IF L_Runtime_OK AND (GVL_TIME_MONOTONIC.Boot_Generation_ID = 0) THEN
    L_Runtime_OK := FALSE;
    L_Error_Code := 4905;
    L_Error_Text := 'Boot generation missing';
END_IF;

IF L_Runtime_OK AND (NOT GVL_STATUS.G_Is_Active_PLC) THEN
    L_Runtime_OK := FALSE;
    L_Error_Code := 5000;
    L_Error_Text := 'Runtime barrier inactive PLC';
END_IF;

IF L_Runtime_OK AND (NOT GVL_PLC_FENCING.PLC_Ownership_Valid) THEN
    L_Runtime_OK := FALSE;
    L_Error_Code := 5010;
    L_Error_Text := 'PLC ownership invalid';
END_IF;

IF L_Runtime_OK AND (NOT GVL_PLC_FENCING.PLC_Semantic_Authority_Valid) THEN
    L_Runtime_OK := FALSE;
    L_Error_Code := 5011;
    L_Error_Text := 'PLC semantic authority invalid';
END_IF;

IF L_Runtime_OK AND GVL_PLC_FENCING.PLC_Forced_Safe_Quarantine THEN
    L_Runtime_OK := FALSE;
    L_Error_Code := 5012;
    L_Error_Text := 'PLC fencing quarantine active';
END_IF;

IF L_Runtime_OK AND GVL_PLC_FENCING.PLC_Lease_Expired THEN
    L_Runtime_OK := FALSE;
    L_Error_Code := 5013;
    L_Error_Text := 'PLC authority lease expired';
END_IF;

IF L_Runtime_OK AND (GVL_PLC_FENCING.PLC_Fencing_Token = 0) THEN
    L_Runtime_OK := FALSE;
    L_Error_Code := 5014;
    L_Error_Text := 'PLC fencing token missing';
END_IF;

IF L_Runtime_OK AND (NOT GVL_TRANSPORT_FRESHNESS.Transport_Freshness_Valid) THEN
    L_Runtime_OK := FALSE;
    L_Error_Code := 5200;
    L_Error_Text := 'Transport freshness invalid';
END_IF;

IF L_Runtime_OK AND (NOT GVL_TRANSPORT_FRESHNESS.Transport_Publication_Allowed) THEN
    L_Runtime_OK := FALSE;
    L_Error_Code := 5201;
    L_Error_Text := 'Transport publication blocked';
END_IF;

IF L_Runtime_OK AND GVL_TRANSPORT_FRESHNESS.Transport_Quarantine_Active THEN
    L_Runtime_OK := FALSE;
    L_Error_Code := 5202;
    L_Error_Text := 'Transport quarantine active';
END_IF;

IF L_Runtime_OK AND GVL_TRANSPORT_FRESHNESS.Transport_Lease_Expired THEN
    L_Runtime_OK := FALSE;
    L_Error_Code := 5203;
    L_Error_Text := 'Transport lease expired';
END_IF;

IF L_Runtime_OK AND GVL_TRANSPORT_FRESHNESS.Transport_Snapshot_Invalid THEN
    L_Runtime_OK := FALSE;
    L_Error_Code := 5204;
    L_Error_Text := 'Transport snapshot invalid';
END_IF;

// Finalized distributed commit continuity.
// Intentionally excludes semantic continuity
// to avoid primordial semantic/runtime recursion.
L_Finalized_Continuity_Healthy :=
    GVL_DISTRIBUTED_SNAPSHOT.Distributed_Publication_Reconciled
    AND GVL_DISTRIBUTED_SNAPSHOT.Distributed_Publication_Freeze_Valid
    AND GVL_DISTRIBUTED_SNAPSHOT.Distributed_Snapshot_Consistent
    AND GVL_DISTRIBUTED_COMMIT.Distributed_Commit_Valid
    AND GVL_DISTRIBUTED_COMMIT.Publication_Prepare_Valid
    AND GVL_DISTRIBUTED_COMMIT.Publication_Commit_Confirmed
    AND NOT GVL_DISTRIBUTED_COMMIT.Peer_Commit_Mismatch
    AND NOT GVL_DISTRIBUTED_COMMIT.Commit_Lease_Expired;

IF L_Runtime_OK
AND NOT L_Finalized_Continuity_Healthy THEN
    L_Runtime_OK := FALSE;
    L_Error_Code := 5300;
    L_Error_Text := 'Finalized continuity invalid';
END_IF;

IF L_Runtime_OK THEN
    IF (GVL_SAFETY_SHUTDOWN.G_Safety_Mode = FIRE)
    AND (GVL_COMMAND_SHADOW.G_Vent_Stop)
    THEN
        L_Runtime_OK := FALSE;
        L_Error_Code := 5003;
        L_Error_Text := 'Impossible fire ventilation state';
    END_IF;
END_IF;

IF L_Runtime_OK THEN
    IF (GVL_SAFETY_SHUTDOWN.G_Safety_Mode = GAS)
    AND (NOT GVL_COMMAND_SHADOW.G_Gas_Valve_Close)
    THEN
        L_Runtime_OK := FALSE;
        L_Error_Code := 5004;
        L_Error_Text := 'Impossible gas valve state';
    END_IF;
END_IF;

GVL_RUNTIME_EPOCH.Runtime_Runtime_Barrier_OK := L_Runtime_OK;
GVL_RUNTIME_EPOCH.Runtime_Snapshot_Valid := L_Runtime_OK;
GVL_RUNTIME_EPOCH.Runtime_PLC_Authority_Valid :=
    GVL_STATUS.G_Is_Active_PLC
    AND GVL_PLC_FENCING.PLC_Semantic_Authority_Valid
    AND GVL_PLC_FENCING.PLC_Ownership_Valid
    AND GVL_TIME_MONOTONIC.Monotonic_Time_Valid
    AND GVL_TRANSPORT_FRESHNESS.Transport_Freshness_Valid
    AND L_Finalized_Continuity_Healthy;

GVL_RUNTIME_EPOCH.Runtime_Last_Validation_Time_MS := L_Now_MS;

IF L_Runtime_OK THEN
    GVL_RUNTIME_EPOCH.Runtime_Epoch := GVL_RUNTIME_EPOCH.Runtime_Epoch + 1;
    GVL_RUNTIME_EPOCH.Runtime_IO_Publication_Allowed := TRUE;
    GVL_RUNTIME_EPOCH.Runtime_Snapshot_Published := TRUE;
    GVL_RUNTIME_EPOCH.Runtime_Last_Error_Code := 0;
    GVL_RUNTIME_EPOCH.Runtime_Last_Error_Text := '';
ELSE
    GVL_RUNTIME_EPOCH.Runtime_Impossible_State_Detected := TRUE;
    GVL_RUNTIME_EPOCH.Runtime_Last_Error_Code := L_Error_Code;
    GVL_RUNTIME_EPOCH.Runtime_Last_Error_Text := L_Error_Text;
    GVL_RUNTIME_EPOCH.Runtime_Barrier_Block_Count := GVL_RUNTIME_EPOCH.Runtime_Barrier_Block_Count + 1;
END_IF;

GVL_RUNTIME_EPOCH.Runtime_Cycle_End_MS := L_Now_MS;
          
END_PROGRAM

PROGRAM PRG_Distributed_Epoch_Linearity_Governor

            IF GVL_TEMPORAL_CAUSALITY_CLOSURE_FABRIC.Temporal_Causality_Closure_Granted
AND NOT GVL_DISTRIBUTED_EPOCH_LINEARITY_FABRIC.Epoch_Rollback_Detected
AND NOT GVL_DISTRIBUTED_EPOCH_LINEARITY_FABRIC.Distributed_Epoch_Fork_Detected
AND NOT GVL_DISTRIBUTED_EPOCH_LINEARITY_FABRIC.Stale_Epoch_Application_Detected THEN

    GVL_DISTRIBUTED_EPOCH_LINEARITY_FABRIC.Distributed_Epoch_Linearity_Valid := TRUE;
    GVL_DISTRIBUTED_EPOCH_LINEARITY_FABRIC.Distributed_Epoch_Linearity_Granted := TRUE;
    GVL_DISTRIBUTED_EPOCH_LINEARITY_FABRIC.Distributed_Epoch_Linearity_Valid_Proof := TRUE;
    GVL_DISTRIBUTED_EPOCH_LINEARITY_FABRIC.Epoch_Timeline_Monotonic := TRUE;
    GVL_DISTRIBUTED_EPOCH_LINEARITY_FABRIC.Cluster_Epoch_Consensus_Stable := TRUE;
END_IF;
          
END_PROGRAM

PROGRAM PRG_PLC_Fencing_Governor
  VAR
    L_Now_MS : UDINT;
    L_Delta_MS : UDINT;
    L_Authority_Valid : BOOL := TRUE;
    L_Error_Code : UDINT := 0;
    L_Error_Text : STRING(160) := '';
  END_VAR

            L_Now_MS := GVL_STATUS.G_System_Time_MS;
L_Authority_Valid := TRUE;
L_Error_Code := 0;
L_Error_Text := '';

// ======================================================
// PLC FENCING GOVERNOR
// ======================================================
// Governs distributed PLC ownership semantics.
// Prevents stale-owner resurrection and split-brain.
// ======================================================

GVL_PLC_FENCING.PLC_Split_Brain_Detected := FALSE;
GVL_PLC_FENCING.PLC_Stale_Owner_Detected := FALSE;
GVL_PLC_FENCING.PLC_Asymmetric_Partition_Detected := FALSE;
GVL_PLC_FENCING.PLC_Forced_Safe_Quarantine := FALSE;

// Active PLC ownership validation.
IF L_Authority_Valid AND (NOT GVL_STATUS.G_Is_Active_PLC) THEN
    L_Authority_Valid := FALSE;
    L_Error_Code := 7001;
    L_Error_Text := 'PLC ownership inactive';
END_IF;

// Lease freshness validation.
L_Delta_MS := L_Now_MS - GVL_PLC_FENCING.PLC_Last_Lease_Refresh_MS;

IF L_Authority_Valid AND GVL_PLC_FENCING.PLC_Lease_Active THEN
    IF L_Delta_MS > GVL_PLC_FENCING.PLC_Lease_Timeout_MS THEN
        L_Authority_Valid := FALSE;
        L_Error_Code := 7002;
        L_Error_Text := 'PLC lease expired';
    END_IF;
END_IF;

// Heartbeat-only ownership is unsafe.
IF L_Authority_Valid AND GVL_PLC_FENCING.PLC_Heartbeat_Only_Mode THEN
    L_Authority_Valid := FALSE;
    L_Error_Code := 7003;
    L_Error_Text := 'Heartbeat-only ownership rejected';
END_IF;

// Publish authoritative fencing state.
IF L_Authority_Valid THEN
    GVL_PLC_FENCING.PLC_Ownership_Epoch := GVL_PLC_FENCING.PLC_Ownership_Epoch + 1;
    GVL_PLC_FENCING.PLC_Fencing_Token := GVL_PLC_FENCING.PLC_Ownership_Epoch;

    GVL_PLC_FENCING.PLC_Ownership_Valid := TRUE;
    GVL_PLC_FENCING.PLC_Semantic_Authority_Valid := TRUE;

    GVL_PLC_FENCING.PLC_Lease_Active := TRUE;
    GVL_PLC_FENCING.PLC_Lease_Expired := FALSE;

    GVL_PLC_FENCING.PLC_Last_Lease_Refresh_MS := L_Now_MS;
    GVL_PLC_FENCING.PLC_Last_Authority_Validation_MS := L_Now_MS;

    GVL_PLC_FENCING.PLC_Last_Error_Code := 0;
    GVL_PLC_FENCING.PLC_Last_Error_Text := '';
ELSE
    GVL_PLC_FENCING.PLC_Ownership_Valid := FALSE;
    GVL_PLC_FENCING.PLC_Semantic_Authority_Valid := FALSE;

    GVL_PLC_FENCING.PLC_Lease_Expired := TRUE;
    GVL_PLC_FENCING.PLC_Forced_Safe_Quarantine := TRUE;

    GVL_PLC_FENCING.PLC_Last_Error_Code := L_Error_Code;
    GVL_PLC_FENCING.PLC_Last_Error_Text := L_Error_Text;

    IF L_Error_Code = 7002 THEN
        GVL_PLC_FENCING.PLC_Stale_Owner_Detected := TRUE;
    END_IF;

    IF L_Error_Code = 7003 THEN
        GVL_PLC_FENCING.PLC_Split_Brain_Detected := TRUE;
        GVL_PLC_FENCING.PLC_Asymmetric_Partition_Detected := TRUE;
    END_IF;

    GVL_PLC_FENCING.PLC_Fencing_Invalidation_Count := GVL_PLC_FENCING.PLC_Fencing_Invalidation_Count + 1;
END_IF;
          
END_PROGRAM

PROGRAM PRG_IO_Read
  VAR
    L_i : INT;
    L_Map_Index : INT;
    L_Glass_Index : INT;
    L_Debounce_Time : TIME := T#100MS;
    L_Manifold_Pressure_Raw : WORD;
    L_Manifold_Current_Raw : WORD;
    L_Filtered_Room_Temp : REAL;
    L_Filtered_Floor_Temp : REAL;
    fbDebounce_Switches : ARRAY[1..GVL_CONSTANTS.C_MAX_LIGHT_ZONES] OF FB_System_Timer;
    fbDebounce_Motion : ARRAY[1..GVL_CONSTANTS.C_MAX_LIGHT_ZONES] OF FB_System_Timer;
    fbDebounce_Security_Open : ARRAY[1..GVL_CONSTANTS.C_MAX_SECURITY_SENSORS] OF FB_System_Timer;
    fbDebounce_Security_Glass : ARRAY[1..GVL_CONSTANTS.C_MAX_SECURITY_SENSORS] OF FB_System_Timer;
    fbDebounce_Flood : ARRAY[1..GVL_CONSTANTS.C_MAX_FLOOD_SENSORS] OF FB_System_Timer;
    fbDebounce_Smoke : ARRAY[1..GVL_CONSTANTS.C_MAX_SMOKE_SENSORS] OF FB_System_Timer;
    fbDebounce_Group_2F : FB_System_Timer;
    fbIO_Watchdog_1 : FB_IO_Module_Watchdog;
    fbIO_Watchdog_2 : FB_IO_Module_Watchdog;
    fbDiagEventManager : FB_Diagnostics_Event_Manager;
    L_IO_Error_Active : BOOL;
    fbCalib_Outdoor_Temp : FB_Sensor_Calibration_Processor;
    fbCalib_Supply_Temps : ARRAY[1..GVL_CONSTANTS.C_MAX_SUPPLY_TEMPS] OF FB_Sensor_Calibration_Processor;
    fbCalib_Room_Temps : ARRAY[1..GVL_CONSTANTS.C_MAX_ZONES] OF FB_Sensor_Calibration_Processor;
    fbCalib_Floor_Temps : ARRAY[1..GVL_CONSTANTS.C_MAX_ZONES] OF FB_Sensor_Calibration_Processor;
    fbCalib_Room_Hum : ARRAY[1..GVL_CONSTANTS.C_MAX_ZONES] OF FB_Sensor_Calibration_Processor;
    fbCalib_Room_CO2 : ARRAY[1..GVL_CONSTANTS.C_MAX_ZONES] OF FB_Sensor_Calibration_Processor;
    fbCalib_Manifold_T_Supply : ARRAY[1..GVL_CONSTANTS.C_MAX_MANIFOLDS] OF FB_Sensor_Calibration_Processor;
    fbCalib_Manifold_T_Return : ARRAY[1..GVL_CONSTANTS.C_MAX_MANIFOLDS] OF FB_Sensor_Calibration_Processor;
    fbCalib_Methane : ARRAY[1..GVL_CONSTANTS.C_MAX_METHANE_SENSORS] OF FB_Sensor_Calibration_Processor;
    fbCalib_CO : ARRAY[1..GVL_CONSTANTS.C_MAX_CO_SENSORS] OF FB_Sensor_Calibration_Processor;
    fbAnalog_Manifold_Pressure : ARRAY[1..GVL_CONSTANTS.C_MAX_MANIFOLDS] OF FB_Sensor_Analog_Processing;
    fbAnalog_Manifold_Current : ARRAY[1..GVL_CONSTANTS.C_MAX_MANIFOLDS] OF FB_Sensor_Analog_Processing;
  END_VAR

            fbIO_Watchdog_1(VI_System_Time_MS := GVL_STATUS.G_System_Time_MS, VI_Module_ID := 1, VI_Heartbeat_Signal := GVL_IO.DI_Module_1_Heartbeat, VI_Timeout_MS := 2000);
fbIO_Watchdog_2(VI_System_Time_MS := GVL_STATUS.G_System_Time_MS, VI_Module_ID := 2, VI_Heartbeat_Signal := GVL_IO.DI_Module_2_Heartbeat, VI_Timeout_MS := 2000);

GVL_STATUS.G_IO_Modules_Online[1] := fbIO_Watchdog_1.VO_Module_Online;
GVL_STATUS.G_IO_Modules_Online[2] := fbIO_Watchdog_2.VO_Module_Online;

L_IO_Error_Active := fbIO_Watchdog_1.VO_Error_Active OR fbIO_Watchdog_2.VO_Error_Active;

fbDiagEventManager(
    VI_Code := 16#E001,
    VI_Severity := 4,
    VI_Active := NOT fbIO_Watchdog_1.VO_Module_Online,
    VI_Timestamp := GVL_STATUS.G_System_Time_MS,
    VI_Source := 1,
    VIO_Events := GVL_STATUS.G_Diagnostics_Events,
    VIO_Count := GVL_STATUS.G_Diagnostics_Count
);

fbDiagEventManager(
    VI_Code := 16#E002,
    VI_Severity := 4,
    VI_Active := NOT fbIO_Watchdog_2.VO_Module_Online,
    VI_Timestamp := GVL_STATUS.G_System_Time_MS,
    VI_Source := 2,
    VIO_Events := GVL_STATUS.G_Diagnostics_Events,
    VIO_Count := GVL_STATUS.G_Diagnostics_Count
);

// Lighting and motion are sized by C_MAX_LIGHT_ZONES.
FOR L_i := 1 TO GVL_CONSTANTS.C_MAX_LIGHT_ZONES DO
    fbDebounce_Switches[L_i](IN := GVL_IO.DI_Lighting_Switches[L_i], PT := L_Debounce_Time, VI_System_Time_MS := GVL_STATUS.G_System_Time_MS);
    GVL_STATE.G_Physical_Switches[L_i] := fbDebounce_Switches[L_i].Q;
    
    fbDebounce_Motion[L_i](IN := GVL_IO.DI_Motion_Sensors[L_i], PT := L_Debounce_Time, VI_System_Time_MS := GVL_STATUS.G_System_Time_MS);
    GVL_STATE.G_Motion_Sensors[L_i] := fbDebounce_Motion[L_i].Q;
END_FOR;

// Socket hardware inputs are propagated instead of being forced to FALSE.
FOR L_i := 1 TO GVL_CONSTANTS.C_MAX_SOCKETS DO
    GVL_STATE.G_Socket_Switches[L_i] := GVL_IO.DI_Socket_Switches[L_i];
END_FOR;

FOR L_i := 1 TO GVL_CONSTANTS.C_MAX_SECURITY_SENSORS DO
    fbDebounce_Security_Open[L_i](IN := GVL_IO.DI_Security_Open[L_i], PT := L_Debounce_Time, VI_System_Time_MS := GVL_STATUS.G_System_Time_MS);
    fbDebounce_Security_Glass[L_i](IN := GVL_IO.DI_Security_Glass[L_i], PT := L_Debounce_Time, VI_System_Time_MS := GVL_STATUS.G_System_Time_MS);
END_FOR;

fbDebounce_Group_2F(IN := GVL_IO.DI_Security_2F_Group, PT := L_Debounce_Time, VI_System_Time_MS := GVL_STATUS.G_System_Time_MS);

FOR L_i := 1 TO GVL_CONSTANTS.C_MAX_DOOR_SENSORS DO
    IF GVL_CONFIG.G_Door_Map[L_i] > 0 AND GVL_CONFIG.G_Door_Map[L_i] <= GVL_CONSTANTS.C_MAX_SECURITY_SENSORS THEN
        GVL_STATE.G_Door_Sensors[L_i] := fbDebounce_Security_Open[GVL_CONFIG.G_Door_Map[L_i]].Q;
    END_IF;
END_FOR;

// Window/opening mapping is limited by C_MAX_ZONES and protected by bounds checks.
FOR L_i := 1 TO GVL_CONSTANTS.C_MAX_ZONES DO
    L_Map_Index := GVL_CONFIG.G_Window_Map[L_i];
    IF L_Map_Index > 0 THEN
        IF L_Map_Index <= GVL_CONSTANTS.C_MAX_SECURITY_SENSORS THEN
            GVL_STATE.G_Window_Sensors[L_i] := fbDebounce_Security_Open[L_Map_Index].Q;
        ELSE
            L_Glass_Index := L_Map_Index - GVL_CONSTANTS.C_MAX_SECURITY_SENSORS;
            IF (L_Glass_Index >= 1) AND (L_Glass_Index <= GVL_CONSTANTS.C_MAX_SECURITY_SENSORS) THEN
                GVL_STATE.G_Window_Sensors[L_i] := fbDebounce_Security_Glass[L_Glass_Index].Q;
            END_IF;
        END_IF;
    END_IF;
END_FOR;
GVL_STATE.G_Window_Sensors[16] := fbDebounce_Group_2F.Q;

FOR L_i := 1 TO GVL_CONSTANTS.C_MAX_FLOOD_SENSORS DO
    fbDebounce_Flood[L_i](IN := GVL_IO.DI_Flood_Sensors[L_i], PT := L_Debounce_Time, VI_System_Time_MS := GVL_STATUS.G_System_Time_MS);
    GVL_STATE.G_Water_Sensors[L_i] := fbDebounce_Flood[L_i].Q;
END_FOR;

FOR L_i := 1 TO GVL_CONSTANTS.C_MAX_SMOKE_SENSORS DO
    fbDebounce_Smoke[L_i](IN := GVL_IO.DI_Smoke_Sensors[L_i], PT := L_Debounce_Time, VI_System_Time_MS := GVL_STATUS.G_System_Time_MS);
    GVL_STATE.G_Smoke_Sensors[L_i] := fbDebounce_Smoke[L_i].Q;
END_FOR;

fbCalib_Outdoor_Temp(
    VI_Raw_Value := GVL_IO.AI_Temp_Outdoor.rValue,
    VI_Record := GVL_CONFIG.G_Calib_Outdoor_Temp
);
GVL_STATE.G_Outdoor_Temp := fbCalib_Outdoor_Temp.VO_Calibrated_Value;

FOR L_i := 1 TO GVL_CONSTANTS.C_MAX_SUPPLY_TEMPS DO
    IF GVL_IO.AI_Supply_Temps[L_i].wStatus = 0 THEN
        fbCalib_Supply_Temps[L_i](
            VI_Raw_Value := GVL_IO.AI_Supply_Temps[L_i].rValue,
            VI_Record := GVL_CONFIG.G_Calib_Supply_Temps[L_i]
        );
        GVL_STATE.G_Supply_Temps[L_i] := fbCalib_Supply_Temps[L_i].VO_Calibrated_Value;
    END_IF;
END_FOR;

// Humidity and CO2 IO/state/calibration arrays are sized by C_MAX_ZONES.
FOR L_i := 1 TO GVL_CONSTANTS.C_MAX_ZONES DO
    fbCalib_Room_Hum[L_i](
        VI_Raw_Value := GVL_IO.AI_Room_Hum[L_i],
        VI_Record := GVL_CONFIG.G_Calib_Humidity[L_i]
    );
    GVL_STATE.G_Room_Hum[L_i] := fbCalib_Room_Hum[L_i].VO_Calibrated_Value;

    fbCalib_Room_CO2[L_i](
        VI_Raw_Value := GVL_IO.AI_Room_CO2[L_i],
        VI_Record := GVL_CONFIG.G_Calib_CO2[L_i]
    );
    GVL_STATE.G_Room_CO2[L_i] := fbCalib_Room_CO2[L_i].VO_Calibrated_Value;
END_FOR;

// Room temperature filtering and range validation
FOR L_i := 1 TO GVL_CONSTANTS.C_MAX_ZONES DO
    fbCalib_Room_Temps[L_i](
        VI_Raw_Value := GVL_IO.AI_Room_Temps[L_i],
        VI_Record := GVL_CONFIG.G_Calib_Room_Temps[L_i]
    );

    IF GVL_STATE.G_Last_Valid_Room_Temps[L_i] = 0.0 THEN
        L_Filtered_Room_Temp := fbCalib_Room_Temps[L_i].VO_Calibrated_Value;
    ELSE
        L_Filtered_Room_Temp := (GVL_STATE.G_Last_Valid_Room_Temps[L_i] * 0.9) + (fbCalib_Room_Temps[L_i].VO_Calibrated_Value * 0.1);
    END_IF;

    IF (L_Filtered_Room_Temp < -50.0) OR (L_Filtered_Room_Temp > 100.0) THEN
        GVL_STATE.G_Temp_Sensor_Fault[L_i] := TRUE;
        GVL_STATE.G_Room_Temps[L_i] := GVL_STATE.G_Last_Valid_Room_Temps[L_i];
        GVL_STATUS.G_Diagnostics.Sensor_Fault := TRUE;
    ELSE
        GVL_STATE.G_Temp_Sensor_Fault[L_i] := FALSE;
        GVL_STATE.G_Room_Temps[L_i] := L_Filtered_Room_Temp;
        GVL_STATE.G_Last_Valid_Room_Temps[L_i] := L_Filtered_Room_Temp;
    END_IF;
END_FOR;

// Floor temperature filtering and range validation
FOR L_i := 1 TO GVL_CONSTANTS.C_MAX_HEATING_CIRCUITS DO
    IF L_i <= GVL_CONSTANTS.C_MAX_ZONES THEN
        fbCalib_Floor_Temps[L_i](
            VI_Raw_Value := GVL_IO.AI_Floor_Temps[L_i],
            VI_Record := GVL_CONFIG.G_Calib_Floor_Temps[L_i]
        );

        IF GVL_STATE.G_Last_Valid_Floor_Temps[L_i] = 0.0 THEN
            L_Filtered_Floor_Temp := fbCalib_Floor_Temps[L_i].VO_Calibrated_Value;
        ELSE
            L_Filtered_Floor_Temp := (GVL_STATE.G_Last_Valid_Floor_Temps[L_i] * 0.9) + (fbCalib_Floor_Temps[L_i].VO_Calibrated_Value * 0.1);
        END_IF;

        IF (L_Filtered_Floor_Temp < -50.0) OR (L_Filtered_Floor_Temp > 100.0) THEN
            GVL_STATE.G_Floor_Temp_Sensor_Fault[L_i] := TRUE;
            GVL_STATE.G_Floor_Temps[L_i] := GVL_STATE.G_Last_Valid_Floor_Temps[L_i];
            GVL_STATUS.G_Diagnostics.Sensor_Fault := TRUE;
        ELSE
            GVL_STATE.G_Floor_Temp_Sensor_Fault[L_i] := FALSE;
            GVL_STATE.G_Floor_Temps[L_i] := L_Filtered_Floor_Temp;
            GVL_STATE.G_Last_Valid_Floor_Temps[L_i] := L_Filtered_Floor_Temp;
        END_IF;
    ELSE
        GVL_STATE.G_Floor_Temp_Sensor_Fault[L_i] := TRUE;
        GVL_STATE.G_Floor_Temps[L_i] := GVL_STATE.G_Last_Valid_Floor_Temps[L_i];
    END_IF;
END_FOR;

GVL_STATUS.G_Diagnostics.Manifold_Pressure_Fault_Active := FALSE;
GVL_STATUS.G_Diagnostics.Manifold_Pressure_First_Fault_Index := 0;
GVL_STATUS.G_Diagnostics.Manifold_Current_Fault_Active := FALSE;
GVL_STATUS.G_Diagnostics.Manifold_Current_First_Fault_Index := 0;
GVL_STATUS.G_Diagnostics.Manifold_Pressure_Fault_Text := '';
GVL_STATUS.G_Diagnostics.Manifold_Current_Fault_Text := '';

FOR L_i := 1 TO GVL_CONSTANTS.C_MAX_MANIFOLDS DO
    IF GVL_IO.AI_Manifold_Pressures[L_i] < 0 THEN
        L_Manifold_Pressure_Raw := 0;
    ELSE
        L_Manifold_Pressure_Raw := INT_TO_WORD(GVL_IO.AI_Manifold_Pressures[L_i]);
    END_IF;

    IF GVL_IO.AI_Manifold_Currents[L_i] < 0 THEN
        L_Manifold_Current_Raw := 0;
    ELSE
        L_Manifold_Current_Raw := INT_TO_WORD(GVL_IO.AI_Manifold_Currents[L_i]);
    END_IF;

    fbAnalog_Manifold_Pressure[L_i](
        VI_Raw_Value := L_Manifold_Pressure_Raw,
        VI_Sensor_Type := 0,
        VI_Min_Scale := 0.0,
        VI_Max_Scale := 10.0,
        VI_Offset := 0.0,
        VI_Multiplier := 1.0,
        VI_Filter_Time_MS := GVL_CONSTANTS.C_MS_IN_SECOND,
        VI_System_Time_MS := GVL_STATUS.G_System_Time_MS,
        VI_Fallback_Mode := 0,
        VI_Default_Value := 0.0
    );
    GVL_STATE.G_Manifold_Pressures[L_i] := fbAnalog_Manifold_Pressure[L_i].VO_Value;
    GVL_STATUS.G_Diagnostics.Manifold_Pressure_Fault[L_i] := fbAnalog_Manifold_Pressure[L_i].VO_Error;
    GVL_STATUS.G_Diagnostics.Manifold_Pressure_Diag_Code[L_i] := fbAnalog_Manifold_Pressure[L_i].VO_Diag_Code;

    fbDiagEventManager(
        VI_Code := GVL_CONFIG.ERR_PRESSURE_OUT_OF_RANGE,
        VI_Severity := 3,
        VI_Active := fbAnalog_Manifold_Pressure[L_i].VO_Error,
        VI_Timestamp := GVL_STATUS.G_System_Time_MS,
        VI_Source := 100 + L_i,
        VIO_Events := GVL_STATUS.G_Diagnostics_Events,
        VIO_Count := GVL_STATUS.G_Diagnostics_Count
    );

    fbAnalog_Manifold_Current[L_i](
        VI_Raw_Value := L_Manifold_Current_Raw,
        VI_Sensor_Type := 0,
        VI_Min_Scale := 0.0,
        VI_Max_Scale := 16.0,
        VI_Offset := 0.0,
        VI_Multiplier := 1.0,
        VI_Filter_Time_MS := GVL_CONSTANTS.C_MS_IN_SECOND,
        VI_System_Time_MS := GVL_STATUS.G_System_Time_MS,
        VI_Fallback_Mode := 0,
        VI_Default_Value := 0.0
    );
    GVL_STATE.G_Manifold_Currents[L_i] := fbAnalog_Manifold_Current[L_i].VO_Value;
    GVL_STATUS.G_Diagnostics.Manifold_Current_Fault[L_i] := fbAnalog_Manifold_Current[L_i].VO_Error;
    GVL_STATUS.G_Diagnostics.Manifold_Current_Diag_Code[L_i] := fbAnalog_Manifold_Current[L_i].VO_Diag_Code;

    fbDiagEventManager(
        VI_Code := GVL_CONFIG.ERR_PUMP_UNDERCURRENT,
        VI_Severity := 3,
        VI_Active := fbAnalog_Manifold_Current[L_i].VO_Error,
        VI_Timestamp := GVL_STATUS.G_System_Time_MS,
        VI_Source := 200 + L_i,
        VIO_Events := GVL_STATUS.G_Diagnostics_Events,
        VIO_Count := GVL_STATUS.G_Diagnostics_Count
    );

    IF GVL_IO.AI_Manifold_Temps_Supply[L_i].wStatus = 0 THEN
        fbCalib_Manifold_T_Supply[L_i](
            VI_Raw_Value := GVL_IO.AI_Manifold_Temps_Supply[L_i].rValue,
            VI_Record := GVL_CONFIG.G_Calib_Manifold_T_Supply[L_i]
        );
        GVL_STATE.G_Manifold_T_Supply[L_i] := fbCalib_Manifold_T_Supply[L_i].VO_Calibrated_Value;
    END_IF;

    fbCalib_Manifold_T_Return[L_i](
        VI_Raw_Value := INT_TO_REAL(GVL_IO.AI_Manifold_Temps_Return[L_i]) / 10.0,
        VI_Record := GVL_CONFIG.G_Calib_Manifold_T_Return[L_i]
    );
    GVL_STATE.G_Manifold_T_Return[L_i] := fbCalib_Manifold_T_Return[L_i].VO_Calibrated_Value;
    GVL_STATE.G_Manifold_End_Switches[L_i] := GVL_IO.DI_Manifold_End_Switches[L_i];

    IF GVL_STATUS.G_Diagnostics.Manifold_Pressure_Fault[L_i] OR GVL_STATUS.G_Diagnostics.Manifold_Current_Fault[L_i] THEN
        GVL_STATUS.G_Diagnostics.Sensor_Fault := TRUE;
        GVL_STATUS.G_Diagnostics.Subsystem_Degraded := TRUE;
    END_IF;

    IF GVL_STATUS.G_Diagnostics.Manifold_Pressure_Fault[L_i] AND GVL_STATUS.G_Diagnostics.Manifold_Current_Fault[L_i] THEN
        GVL_STATUS.G_Diagnostics.Manifold_Pressure_Fault_Text := 'Correlated pressure/current fault detected';
        GVL_STATUS.G_Diagnostics.Manifold_Current_Fault_Text := 'Correlated pressure/current fault detected';
    ELSIF GVL_STATUS.G_Diagnostics.Manifold_Pressure_Fault[L_i] AND (GVL_STATUS.G_Diagnostics.Manifold_Pressure_Fault_Text = '') THEN
        GVL_STATUS.G_Diagnostics.Manifold_Pressure_Fault_Text := 'Pressure sensor fault detected';
    ELSIF GVL_STATUS.G_Diagnostics.Manifold_Current_Fault[L_i] AND (GVL_STATUS.G_Diagnostics.Manifold_Current_Fault_Text = '') THEN
        GVL_STATUS.G_Diagnostics.Manifold_Current_Fault_Text := 'Current sensor fault detected';
    END_IF;
END_FOR;

FOR L_i := 1 TO GVL_CONSTANTS.C_MAX_METHANE_SENSORS DO
    IF GVL_IO.AI_Methane_LEL[L_i].wStatus = 0 THEN
        fbCalib_Methane[L_i](
            VI_Raw_Value := GVL_IO.AI_Methane_LEL[L_i].rValue,
            VI_Record := GVL_CONFIG.G_Calib_Methane[L_i]
        );
        GVL_STATE.G_Methane_Sensors[L_i] := fbCalib_Methane[L_i].VO_Calibrated_Value;
    END_IF;

    fbDiagEventManager(
        VI_Code := 16#E003,
        VI_Severity := 3,
        VI_Active := GVL_IO.AI_Methane_LEL[L_i].wStatus <> 0,
        VI_Timestamp := GVL_STATUS.G_System_Time_MS,
        VI_Source := 300 + L_i,
        VIO_Events := GVL_STATUS.G_Diagnostics_Events,
        VIO_Count := GVL_STATUS.G_Diagnostics_Count
    );
END_FOR;

FOR L_i := 1 TO GVL_CONSTANTS.C_MAX_CO_SENSORS DO
    fbCalib_CO[L_i](
        VI_Raw_Value := GVL_IO.AI_CO_PPM[L_i],
        VI_Record := GVL_CONFIG.G_Calib_CO[L_i]
    );
    GVL_STATE.G_CO_Sensors[L_i] := fbCalib_CO[L_i].VO_Calibrated_Value;
END_FOR;

GVL_STATE.G_DHW_Temp := GVL_IO.AI_DHW_Temp;
GVL_STATE.G_DHW_Pressure := GVL_IO.AI_DHW_Pressure;

GVL_STATE.G_Water_Zone_Open_FB := GVL_IO.DI_Water_Zone_Open_FB;
GVL_STATE.G_Water_Zone_Close_FB := GVL_IO.DI_Water_Zone_Close_FB;

// >>> BULK_SYNC_ANCHOR: PRG_IO_Read <<<
          
END_PROGRAM

PROGRAM PRG_System_Access_Maintenance
  VAR
    fbLogEvent : FB_LogEvent;
    L_Dangerous_Action_Armed : BOOL;
    L_Dangerous_Action_Deadline_MS : UDINT;
    L_Maintenance_Apply_Intent : BOOL;
    L_User_Access_Denied_Prev : BOOL;
  END_VAR

            L_Maintenance_Apply_Intent := FALSE;

// Dangerous action request
IF GVL_COMMAND.CMD_Dangerous_Action_Request AND (GVL_COMMAND.CMD_User_Access_Level >= 2) THEN
    IF NOT L_Dangerous_Action_Armed THEN
        fbLogEvent(
            VI_Event_Type := 8,
            VI_Timestamp := GVL_TIME_SERVICE.G_Now_MS,
            VI_Param1 := TO_UDINT(GVL_COMMAND.CMD_User_Access_Level),
            VI_Param2 := 1
        );
    END_IF;

    L_Dangerous_Action_Armed := TRUE;
    L_Dangerous_Action_Deadline_MS := GVL_TIME_SERVICE.G_Now_MS + 15000;

    GVL_STATUS.G_Diagnostics.Dangerous_Action_Pending_Confirm := TRUE;
    GVL_STATUS.G_Diagnostics.Dangerous_Action_Confirm_Deadline_MS := L_Dangerous_Action_Deadline_MS;
    GVL_STATUS.G_Diagnostics.Dangerous_Action_Confirm_Text := 'Подтвердите опасное действие в течение 15 секунд';
END_IF;

// Timeout
IF L_Dangerous_Action_Armed AND (GVL_TIME_SERVICE.G_Now_MS > L_Dangerous_Action_Deadline_MS) THEN
    L_Dangerous_Action_Armed := FALSE;
    GVL_STATUS.G_Diagnostics.Dangerous_Action_Pending_Confirm := FALSE;
    GVL_STATUS.G_Diagnostics.Dangerous_Action_Confirm_Text := 'Окно подтверждения истекло';
END_IF;

// Confirm
IF GVL_COMMAND.CMD_Dangerous_Action_Confirm AND
   L_Dangerous_Action_Armed AND
   (GVL_COMMAND.CMD_User_Access_Level >= 2) THEN

    L_Maintenance_Apply_Intent := TRUE;

    fbLogEvent(
        VI_Event_Type := 9,
        VI_Timestamp := GVL_TIME_SERVICE.G_Now_MS,
        VI_Param1 := TO_UDINT(GVL_COMMAND.CMD_User_Access_Level),
        VI_Param2 := 1
    );

    L_Dangerous_Action_Armed := FALSE;
    GVL_STATUS.G_Diagnostics.Dangerous_Action_Pending_Confirm := FALSE;
    GVL_STATUS.G_Diagnostics.Dangerous_Action_Confirm_Text := 'Опасное действие подтверждено оператором';
END_IF;

// Apply maintenance
IF L_Maintenance_Apply_Intent THEN
    GVL_CONFIG.G_DHW_Heating_Pump_In_Service := GVL_COMMAND.CMD_Set_DHW_Heating_Pump_In_Service;
    GVL_CONFIG.G_DHW_Circ_Pump_In_Service := GVL_COMMAND.CMD_Set_DHW_Circ_Pump_In_Service;
END_IF;

// Access enforcement
GVL_STATUS.G_Diagnostics.User_Access_Level_Active := GVL_COMMAND.CMD_User_Access_Level;
GVL_STATUS.G_Diagnostics.User_Access_Denied := FALSE;

IF GVL_COMMAND.CMD_Dangerous_Action_Request OR GVL_COMMAND.CMD_Dangerous_Action_Confirm THEN
    IF GVL_COMMAND.CMD_User_Access_Level < 2 THEN
        IF NOT L_User_Access_Denied_Prev THEN
            fbLogEvent(
                VI_Event_Type := 10,
                VI_Timestamp := GVL_TIME_SERVICE.G_Now_MS,
                VI_Param1 := TO_UDINT(GVL_COMMAND.CMD_User_Access_Level),
                VI_Param2 := 2
            );
        END_IF;

        GVL_STATUS.G_Diagnostics.User_Access_Denied := TRUE;
        GVL_STATUS.G_Diagnostics.Operator_Action_Blocked := TRUE;
    END_IF;
END_IF;

L_User_Access_Denied_Prev := GVL_STATUS.G_Diagnostics.User_Access_Denied;
          
END_PROGRAM

PROGRAM PRG_System_Health
  VAR
    fbSystemHealthOrchestrator : FB_System_Health_Orchestrator;
  END_VAR

            // Centralized Health execution (Phase 5)
fbSystemHealthOrchestrator(
    VO_First_Fault_Active => GVL_SYSTEM_HEALTH.G_First_Fault_Active,
    VO_First_Fault_Type => GVL_SYSTEM_HEALTH.G_First_Fault_Type,
    VO_First_Fault_Source => GVL_SYSTEM_HEALTH.G_First_Fault_Source,
    VO_System_Severity => GVL_SYSTEM_HEALTH.G_System_Severity,
    VO_Root_Cause => GVL_SYSTEM_HEALTH.G_Root_Cause,
    VO_Watchdog_Fault => GVL_SYSTEM_HEALTH.G_Watchdog_Fault
);
          
END_PROGRAM

PROGRAM PRG_Access
  VAR
    fbProjection : FB_Access_Output_Projection;
    L_Mode : E_Safety_Mode;
    L_Now_MS : UDINT;
    L_Elapsed_MS : UDINT;
    L_Pulse_MS : UDINT;
    L_Distributed_Execute_Allowed : BOOL;
    L_Distributed_Access_Allowed : BOOL;
    L_Lock_1_Open : BOOL;
    L_Lock_1_Close : BOOL;
    L_Lock_2_Open : BOOL;
    L_Lock_2_Close : BOOL;
    L_Gate_Open : BOOL;
    L_Wicket_Open : BOOL;
    L_Prev_Lock_1_Open : BOOL;
    L_Prev_Lock_1_Close : BOOL;
    L_Prev_Lock_2_Open : BOOL;
    L_Prev_Lock_2_Close : BOOL;
    L_Prev_Gate_Open : BOOL;
    L_Prev_Wicket_Open : BOOL;
    L_Pulse_Lock_1_Open : BOOL;
    L_Pulse_Lock_1_Close : BOOL;
    L_Pulse_Lock_2_Open : BOOL;
    L_Pulse_Lock_2_Close : BOOL;
    L_Pulse_Gate_Open : BOOL;
    L_Pulse_Wicket_Open : BOOL;
    L_Start_Lock_1_Open_MS : UDINT;
    L_Start_Lock_1_Close_MS : UDINT;
    L_Start_Lock_2_Open_MS : UDINT;
    L_Start_Lock_2_Close_MS : UDINT;
    L_Start_Gate_Open_MS : UDINT;
    L_Start_Wicket_Open_MS : UDINT;
  END_VAR

            L_Mode := GVL_SAFETY_SHUTDOWN.G_Safety_Mode;
L_Now_MS := GVL_STATUS.G_System_Time_MS;

// Distributed runtime governance.
// FIRE/GAS emergency semantics remain authoritative.
L_Distributed_Execute_Allowed :=
    GVL_Distributed_Execution_Gates.G_Can_Execute;

L_Distributed_Access_Allowed :=
    GVL_Distributed_Execution_Gates.G_Can_Own_Projection;

IF (L_Mode <> FIRE)
   AND (L_Mode <> GAS)
   AND (
        NOT L_Distributed_Execute_Allowed
        OR NOT L_Distributed_Access_Allowed
       ) THEN

    fbProjection(
        VI_Lock_1_Open := FALSE,
        VI_Lock_1_Close := FALSE,
        VI_Lock_2_Open := FALSE,
        VI_Lock_2_Close := FALSE,
        VI_Gate_Open := FALSE,
        VI_Wicket_Open := FALSE
    );

    RETURN;
END_IF;

// Load pulse duration from config with safety clamp
L_Pulse_MS := GVL_CONFIG.G_Access_Pulse_MS;
IF L_Pulse_MS < 100 THEN
    L_Pulse_MS := 100;
ELSIF L_Pulse_MS > 5000 THEN
    L_Pulse_MS := 5000;
END_IF;

L_Lock_1_Open := FALSE;
L_Lock_1_Close := FALSE;
L_Lock_2_Open := FALSE;
L_Lock_2_Close := FALSE;
L_Gate_Open := FALSE;
L_Wicket_Open := FALSE;

CASE L_Mode OF
    FIRE:
        L_Lock_1_Open := GVL_COMMAND_SHADOW.G_Lock_1_Open;
        L_Lock_2_Open := GVL_COMMAND_SHADOW.G_Lock_2_Open;
        L_Gate_Open := GVL_COMMAND_SHADOW.G_Gate_Open;
        L_Wicket_Open := GVL_COMMAND_SHADOW.G_Wicket_Open;

        L_Pulse_Lock_1_Open := FALSE;
        L_Pulse_Lock_1_Close := FALSE;
        L_Pulse_Lock_2_Open := FALSE;
        L_Pulse_Lock_2_Close := FALSE;
        L_Pulse_Gate_Open := FALSE;
        L_Pulse_Wicket_Open := FALSE;

        L_Prev_Lock_1_Open := GVL_COMMAND_SHADOW.G_Lock_1_Open;
        L_Prev_Lock_1_Close := GVL_COMMAND_SHADOW.G_Lock_1_Close;
        L_Prev_Lock_2_Open := GVL_COMMAND_SHADOW.G_Lock_2_Open;
        L_Prev_Lock_2_Close := GVL_COMMAND_SHADOW.G_Lock_2_Close;
        L_Prev_Gate_Open := GVL_COMMAND_SHADOW.G_Gate_Open;
        L_Prev_Wicket_Open := GVL_COMMAND_SHADOW.G_Wicket_Open;

    GAS:
        L_Gate_Open := GVL_COMMAND_SHADOW.G_Gate_Open;

        IF GVL_COMMAND_SHADOW.G_Lock_1_Open AND NOT L_Prev_Lock_1_Open THEN
            L_Pulse_Lock_1_Open := TRUE;
            L_Start_Lock_1_Open_MS := L_Now_MS;
        END_IF;
        IF GVL_COMMAND_SHADOW.G_Lock_2_Open AND NOT L_Prev_Lock_2_Open THEN
            L_Pulse_Lock_2_Open := TRUE;
            L_Start_Lock_2_Open_MS := L_Now_MS;
        END_IF;
        IF GVL_COMMAND_SHADOW.G_Wicket_Open AND NOT L_Prev_Wicket_Open THEN
            L_Pulse_Wicket_Open := TRUE;
            L_Start_Wicket_Open_MS := L_Now_MS;
        END_IF;

        IF L_Pulse_Lock_1_Open THEN
            L_Elapsed_MS := SEL(L_Now_MS >= L_Start_Lock_1_Open_MS, L_Now_MS - L_Start_Lock_1_Open_MS, (4294967295 - L_Start_Lock_1_Open_MS) + L_Now_MS + 1);
            IF L_Elapsed_MS < L_Pulse_MS THEN
                L_Lock_1_Open := TRUE;
            ELSE
                L_Pulse_Lock_1_Open := FALSE;
            END_IF;
        END_IF;

        IF L_Pulse_Lock_2_Open THEN
            L_Elapsed_MS := SEL(L_Now_MS >= L_Start_Lock_2_Open_MS, L_Now_MS - L_Start_Lock_2_Open_MS, (4294967295 - L_Start_Lock_2_Open_MS) + L_Now_MS + 1);
            IF L_Elapsed_MS < L_Pulse_MS THEN
                L_Lock_2_Open := TRUE;
            ELSE
                L_Pulse_Lock_2_Open := FALSE;
            END_IF;
        END_IF;

        IF L_Pulse_Wicket_Open THEN
            L_Elapsed_MS := SEL(L_Now_MS >= L_Start_Wicket_Open_MS, L_Now_MS - L_Start_Wicket_Open_MS, (4294967295 - L_Start_Wicket_Open_MS) + L_Now_MS + 1);
            IF L_Elapsed_MS < L_Pulse_MS THEN
                L_Wicket_Open := TRUE;
            ELSE
                L_Pulse_Wicket_Open := FALSE;
            END_IF;
        END_IF;

        L_Prev_Lock_1_Open := GVL_COMMAND_SHADOW.G_Lock_1_Open;
        L_Prev_Lock_1_Close := GVL_COMMAND_SHADOW.G_Lock_1_Close;
        L_Prev_Lock_2_Open := GVL_COMMAND_SHADOW.G_Lock_2_Open;
        L_Prev_Lock_2_Close := GVL_COMMAND_SHADOW.G_Lock_2_Close;
        L_Prev_Gate_Open := GVL_COMMAND_SHADOW.G_Gate_Open;
        L_Prev_Wicket_Open := GVL_COMMAND_SHADOW.G_Wicket_Open;

ELSE
        IF GVL_COMMAND_SHADOW.G_Lock_1_Open AND NOT L_Prev_Lock_1_Open THEN
            L_Pulse_Lock_1_Open := TRUE;
            L_Start_Lock_1_Open_MS := L_Now_MS;
        END_IF;
        IF GVL_COMMAND_SHADOW.G_Lock_1_Close AND NOT L_Prev_Lock_1_Close THEN
            L_Pulse_Lock_1_Close := TRUE;
            L_Start_Lock_1_Close_MS := L_Now_MS;
        END_IF;
        IF GVL_COMMAND_SHADOW.G_Lock_2_Open AND NOT L_Prev_Lock_2_Open THEN
            L_Pulse_Lock_2_Open := TRUE;
            L_Start_Lock_2_Open_MS := L_Now_MS;
        END_IF;
        IF GVL_COMMAND_SHADOW.G_Lock_2_Close AND NOT L_Prev_Lock_2_Close THEN
            L_Pulse_Lock_2_Close := TRUE;
            L_Start_Lock_2_Close_MS := L_Now_MS;
        END_IF;
        IF GVL_COMMAND_SHADOW.G_Gate_Open AND NOT L_Prev_Gate_Open THEN
            L_Pulse_Gate_Open := TRUE;
            L_Start_Gate_Open_MS := L_Now_MS;
        END_IF;
        IF GVL_COMMAND_SHADOW.G_Wicket_Open AND NOT L_Prev_Wicket_Open THEN
            L_Pulse_Wicket_Open := TRUE;
            L_Start_Wicket_Open_MS := L_Now_MS;
        END_IF;

        IF L_Pulse_Lock_1_Open THEN
            L_Elapsed_MS := SEL(L_Now_MS >= L_Start_Lock_1_Open_MS, L_Now_MS - L_Start_Lock_1_Open_MS, (4294967295 - L_Start_Lock_1_Open_MS) + L_Now_MS + 1);
            IF L_Elapsed_MS < L_Pulse_MS THEN
                L_Lock_1_Open := TRUE;
            ELSE
                L_Pulse_Lock_1_Open := FALSE;
            END_IF;
        END_IF;

        IF L_Pulse_Lock_1_Close THEN
            L_Elapsed_MS := SEL(L_Now_MS >= L_Start_Lock_1_Close_MS, L_Now_MS - L_Start_Lock_1_Close_MS, (4294967295 - L_Start_Lock_1_Close_MS) + L_Now_MS + 1);
            IF L_Elapsed_MS < L_Pulse_MS THEN
                L_Lock_1_Close := TRUE;
            ELSE
                L_Pulse_Lock_1_Close := FALSE;
            END_IF;
        END_IF;

        IF L_Pulse_Lock_2_Open THEN
            L_Elapsed_MS := SEL(L_Now_MS >= L_Start_Lock_2_Open_MS, L_Now_MS - L_Start_Lock_2_Open_MS, (4294967295 - L_Start_Lock_2_Open_MS) + L_Now_MS + 1);
            IF L_Elapsed_MS < L_Pulse_MS THEN
                L_Lock_2_Open := TRUE;
            ELSE
                L_Pulse_Lock_2_Open := FALSE;
            END_IF;
        END_IF;

        IF L_Pulse_Lock_2_Close THEN
            L_Elapsed_MS := SEL(L_Now_MS >= L_Start_Lock_2_Close_MS, L_Now_MS - L_Start_Lock_2_Close_MS, (4294967295 - L_Start_Lock_2_Close_MS) + L_Now_MS + 1);
            IF L_Elapsed_MS < L_Pulse_MS THEN
                L_Lock_2_Close := TRUE;
            ELSE
                L_Pulse_Lock_2_Close := FALSE;
            END_IF;
        END_IF;

        IF L_Pulse_Gate_Open THEN
            L_Elapsed_MS := SEL(L_Now_MS >= L_Start_Gate_Open_MS, L_Now_MS - L_Start_Gate_Open_MS, (4294967295 - L_Start_Gate_Open_MS) + L_Now_MS + 1);
            IF L_Elapsed_MS < L_Pulse_MS THEN
                L_Gate_Open := TRUE;
            ELSE
                L_Pulse_Gate_Open := FALSE;
            END_IF;
        END_IF;

        IF L_Pulse_Wicket_Open THEN
            L_Elapsed_MS := SEL(L_Now_MS >= L_Start_Wicket_Open_MS, L_Now_MS - L_Start_Wicket_Open_MS, (4294967295 - L_Start_Wicket_Open_MS) + L_Now_MS + 1);
            IF L_Elapsed_MS < L_Pulse_MS THEN
                L_Wicket_Open := TRUE;
            ELSE
                L_Pulse_Wicket_Open := FALSE;
            END_IF;
        END_IF;

        L_Prev_Lock_1_Open := GVL_COMMAND_SHADOW.G_Lock_1_Open;
        L_Prev_Lock_1_Close := GVL_COMMAND_SHADOW.G_Lock_1_Close;
        L_Prev_Lock_2_Open := GVL_COMMAND_SHADOW.G_Lock_2_Open;
        L_Prev_Lock_2_Close := GVL_COMMAND_SHADOW.G_Lock_2_Close;
        L_Prev_Gate_Open := GVL_COMMAND_SHADOW.G_Gate_Open;
        L_Prev_Wicket_Open := GVL_COMMAND_SHADOW.G_Wicket_Open;
END_CASE;

fbProjection(
    VI_Lock_1_Open := L_Lock_1_Open,
    VI_Lock_1_Close := L_Lock_1_Close,
    VI_Lock_2_Open := L_Lock_2_Open,
    VI_Lock_2_Close := L_Lock_2_Close,
    VI_Gate_Open := L_Gate_Open,
    VI_Wicket_Open := L_Wicket_Open
);

// >>> BULK_SYNC_ANCHOR: PRG_Access <<<
          
END_PROGRAM

PROGRAM PRG_System_Intent
  VAR
    fbSystemIntentPublisher : FB_System_Intent_Publisher;
    L_Gateway_Writes_Allowed : BOOL;
  END_VAR

            // Extracted from PRG_System (Phase 5A).
// Idempotent projection: safe to run while legacy call still exists.
L_Gateway_Writes_Allowed :=
    NOT GVL_STATUS.G_Diagnostics.Dangerous_Action_Pending_Confirm AND
    NOT GVL_STATUS.G_Diagnostics.Operator_Action_Blocked AND
    NOT GVL_STATUS.G_Diagnostics.User_Access_Denied;

fbSystemIntentPublisher(
    VI_System_Time_MS := GVL_TIME_SERVICE.G_Now_MS,
    VI_Gateway_Writes_Allowed := L_Gateway_Writes_Allowed
);
          
END_PROGRAM

PROGRAM PRG_Modbus_RTU_Driver
  VAR
    FB_RTU_Driver : FB_Modbus_RTU_Driver;
  END_VAR

            // ======================================================
// MODBUS RTU DRIVER EXECUTION
// ======================================================
// Runtime execution wrapper for the RTU driver FB.
//
// Driver_Attached is a configuration/HMI decision and must not depend
// on runtime bridge state.
// ======================================================

FB_RTU_Driver(
    VI_Enable := GVL_CONFIG.G_OpenTherm_Enabled,
    VI_Driver_Attached := GVL_CONFIG.G_Modbus_RTU_Driver_Attached,
    VI_System_Time_MS := GVL_STATUS.G_System_Time_MS
);
          
END_PROGRAM

PROGRAM PRG_Physical_SafeState_Lattice_Governor
  VAR
    L_Now_MS : UDINT;
    L_Valid : BOOL := TRUE;
  END_VAR

            L_Now_MS := GVL_STATUS.G_System_Time_MS;

GVL_PHYSICAL_SAFESTATE_LATTICE_FABRIC.Physical_SafeState_Lattice_Valid := FALSE;
GVL_PHYSICAL_SAFESTATE_LATTICE_FABRIC.Physical_SafeState_Lattice_Granted := FALSE;
GVL_PHYSICAL_SAFESTATE_LATTICE_FABRIC.Physical_SafeState_Lattice_Quarantine_Active := TRUE;

IF NOT GVL_GOVERNANCE_PUBLICATION_BINDING_FABRIC.Governance_Publication_Binding_Granted THEN
    L_Valid := FALSE;
END_IF;

IF GVL_PHYSICAL_SAFESTATE_LATTICE_FABRIC.SafeState_Ambiguity_Detected
OR GVL_PHYSICAL_SAFESTATE_LATTICE_FABRIC.Partial_SafeState_Asymmetry_Detected
OR GVL_PHYSICAL_SAFESTATE_LATTICE_FABRIC.Physical_SafeState_Deadlock_Detected
OR GVL_PHYSICAL_SAFESTATE_LATTICE_FABRIC.Unsafe_SafeState_Topology_Detected
OR GVL_PHYSICAL_SAFESTATE_LATTICE_FABRIC.Residual_Unsafe_Actuation_Detected
OR GVL_PHYSICAL_SAFESTATE_LATTICE_FABRIC.SafeState_Energy_Leakage_Detected THEN
    L_Valid := FALSE;
END_IF;

IF L_Valid THEN
    GVL_PHYSICAL_SAFESTATE_LATTICE_FABRIC.Physical_SafeState_Lattice_Valid := TRUE;
    GVL_PHYSICAL_SAFESTATE_LATTICE_FABRIC.Physical_SafeState_Lattice_Granted := TRUE;
    GVL_PHYSICAL_SAFESTATE_LATTICE_FABRIC.Physical_SafeState_Lattice_Quarantine_Active := FALSE;

    GVL_PHYSICAL_SAFESTATE_LATTICE_FABRIC.Canonical_SafeState_Topology_Valid := TRUE;
    GVL_PHYSICAL_SAFESTATE_LATTICE_FABRIC.Physical_SafeState_Lattice_Coherent := TRUE;
    GVL_PHYSICAL_SAFESTATE_LATTICE_FABRIC.Deterministic_FailSafe_Convergence_Granted := TRUE;

    GVL_PHYSICAL_SAFESTATE_LATTICE_FABRIC.Physical_SafeState_Lattice_Epoch :=
        GVL_GOVERNANCE_PUBLICATION_BINDING_FABRIC.Governance_Publication_Binding_Epoch;

    GVL_PHYSICAL_SAFESTATE_LATTICE_FABRIC.Physical_SafeState_Lattice_Epoch_Coherent := TRUE;
    GVL_PHYSICAL_SAFESTATE_LATTICE_FABRIC.Physical_SafeState_Lattice_Last_Update_MS := L_Now_MS;
    GVL_PHYSICAL_SAFESTATE_LATTICE_FABRIC.Physical_SafeState_Lattice_Lease_Expired := FALSE;
END_IF;
          
END_PROGRAM

PROGRAM PRG_HMI_Dashboard
  VAR
    L_i : INT;
  END_VAR

            // ======================================================
// HEATING CONFIDENCE
// ======================================================
GVL_HMI.G_HMI_Heating_Confidence := GVL_STATE.G_Heating_Confidence;
GVL_HMI.G_HMI_Heating_Confidence_Percent := REAL_TO_INT(GVL_STATE.G_Heating_Confidence * 100.0);

// ======================================================
// HEATING ROOT CAUSE
// ======================================================
GVL_HMI.G_HMI_Heating_Reason_Code := GVL_STATE.G_Heating_Confidence_Reason_Code;
GVL_HMI.G_HMI_Heating_Status_Text := GVL_STATE.G_Heating_Confidence_Reason_Text;

// ======================================================
// HEATING STATUS LEVEL
// ======================================================
IF GVL_STATE.G_Heating_Confidence > 0.8 THEN
    GVL_HMI.G_HMI_Heating_Status_Level := 0;
ELSIF GVL_STATE.G_Heating_Confidence > 0.5 THEN
    GVL_HMI.G_HMI_Heating_Status_Level := 1;
ELSE
    GVL_HMI.G_HMI_Heating_Status_Level := 2;
END_IF;

// ======================================================
// CASCADE SEMANTIC STATE
// ======================================================
GVL_HMI.G_HMI_Heating_Cascade_Available :=
    GVL_STATE.G_Heating_Cascade_Available;

GVL_HMI.G_HMI_Heating_Cascade_Degraded :=
    GVL_STATE.G_Heating_Cascade_Degraded;

GVL_HMI.G_HMI_Heating_Cascade_Partial_Capacity :=
    GVL_STATE.G_Heating_Cascade_Partial_Capacity;

GVL_HMI.G_HMI_Heating_Cascade_No_Flame :=
    GVL_STATE.G_Heating_Cascade_No_Flame;

GVL_HMI.G_HMI_Heating_Cascade_Transport_Degraded :=
    GVL_STATE.G_Heating_Cascade_Transport_Degraded;

GVL_HMI.G_HMI_Heating_Cascade_Ignition_Timeout :=
    GVL_STATE.G_Heating_Cascade_Ignition_Timeout;

GVL_HMI.G_HMI_Heating_Cascade_Active_Boilers :=
    GVL_STATE.G_Heating_Cascade_Active_Boilers;

GVL_HMI.G_HMI_Heating_Cascade_Available_Boilers :=
    GVL_STATE.G_Heating_Cascade_Available_Boilers;

// ======================================================
// OPENTHERM SEMANTIC STATE
// ======================================================
FOR L_i := 1 TO GVL_CONSTANTS.C_MAX_BOILERS DO

    GVL_HMI.G_HMI_Boiler_OT_Online[L_i] :=
        GVL_STATE.G_Boiler_OT_Online[L_i];

    GVL_HMI.G_HMI_Boiler_OT_Command_Ack[L_i] :=
        GVL_STATE.G_Boiler_OT_Command_Ack[L_i];

    GVL_HMI.G_HMI_Boiler_OT_Command_Timeout[L_i] :=
        GVL_STATE.G_Boiler_OT_Command_Timeout[L_i];

    GVL_HMI.G_HMI_Boiler_OT_Heartbeat_Timeout[L_i] :=
        GVL_STATE.G_Boiler_OT_Heartbeat_Timeout[L_i];

    GVL_HMI.G_HMI_Boiler_OT_Adapter_Error[L_i] :=
        GVL_STATE.G_Boiler_OT_Adapter_Error[L_i];

    GVL_HMI.G_HMI_Boiler_OT_Heartbeat_Age_MS[L_i] :=
        GVL_STATE.G_Boiler_OT_Heartbeat_Age_MS[L_i];

    GVL_HMI.G_HMI_Boiler_OT_Command_Age_MS[L_i] :=
        GVL_STATE.G_Boiler_OT_Command_Age_MS[L_i];

    GVL_HMI.G_HMI_Boiler_OT_Adapter_State[L_i] :=
        GVL_STATE.G_Boiler_OT_Adapter_State[L_i];

    GVL_HMI.G_HMI_Boiler_OT_Error_State[L_i] :=
        GVL_STATE.G_Boiler_OT_Error_State[L_i];

END_FOR;

// ======================================================
// PREDICTIVE FLAGS
// ======================================================
FOR L_i := 1 TO GVL_CONSTANTS.C_MAX_MANIFOLDS DO
    GVL_HMI.G_HMI_Heating_Predictive_Pressure_Drop[L_i] :=
        GVL_STATE.G_Predictive_Pump_Pressure_Drop[L_i];

    GVL_HMI.G_HMI_Heating_Predictive_Current_Rise[L_i] :=
        GVL_STATE.G_Predictive_Pump_Current_Rise[L_i];
END_FOR;
          
END_PROGRAM

PROGRAM PRG_Config_Manager
  VAR
    L_Error : BOOL;
    L_Index : INT;
  END_VAR

            L_Error := FALSE;
GVL_CONFIG_VALIDATION.G_Config_Auto_Corrected := FALSE;
GVL_CONFIG_CONTROL.G_Apply_Done := FALSE;
GVL_CONFIG_CONTROL.G_Rollback_Done := FALSE;

IF NOT GVL_CONFIG_SIMULATION.G_Simulation_Result_OK THEN
    GVL_CONFIG_CONTROL.G_Apply_Request := FALSE;
END_IF;

// ===== SIZE VALIDATION =====
IF GVL_SYSTEM_SIZE_CONFIG.G_Active_Heating_Circuits < 1 OR GVL_SYSTEM_SIZE_CONFIG.G_Active_Heating_Circuits > GVL_CONSTANTS.C_MAX_HEATING_CIRCUITS THEN
    GVL_SYSTEM_SIZE_CONFIG.G_Active_Heating_Circuits := GVL_CONSTANTS.C_MAX_HEATING_CIRCUITS;
    L_Error := TRUE;
END_IF;

IF GVL_SYSTEM_SIZE_CONFIG.G_Active_Water_Zones < 1 OR GVL_SYSTEM_SIZE_CONFIG.G_Active_Water_Zones > GVL_CONSTANTS.C_MAX_WATER_ZONES THEN
    GVL_SYSTEM_SIZE_CONFIG.G_Active_Water_Zones := GVL_CONSTANTS.C_MAX_WATER_ZONES;
    L_Error := TRUE;
END_IF;

IF GVL_SYSTEM_SIZE_CONFIG.G_Active_Light_Zones < 1 OR GVL_SYSTEM_SIZE_CONFIG.G_Active_Light_Zones > GVL_CONSTANTS.C_MAX_LIGHT_ZONES THEN
    GVL_SYSTEM_SIZE_CONFIG.G_Active_Light_Zones := GVL_CONSTANTS.C_MAX_LIGHT_ZONES;
    L_Error := TRUE;
END_IF;

// ===== EXISTING VALIDATION =====
IF GVL_INPUT_VALIDATION_CONFIG.G_Reputation_Learning_Rate < 0.0 OR GVL_INPUT_VALIDATION_CONFIG.G_Reputation_Learning_Rate > 1.0 THEN
    GVL_INPUT_VALIDATION_CONFIG.G_Reputation_Learning_Rate := 0.05;
    L_Error := TRUE;
END_IF;

// ===== APPLY (unchanged) =====
IF GVL_CONFIG_CONTROL.G_Apply_Request AND GVL_CONFIG_CONTROL.G_Apply_Confirm THEN
    GVL_CONFIG_CONTROL.BCK_Reputation_Learning_Rate := GVL_INPUT_VALIDATION_CONFIG.G_Reputation_Learning_Rate;
    GVL_INPUT_VALIDATION_CONFIG.G_Reputation_Learning_Rate := GVL_CONFIG_CONTROL.STG_Reputation_Learning_Rate;

    GVL_CONFIG_CONTROL.G_Config_Version := GVL_CONFIG_CONTROL.G_Config_Version + 1;

    L_Index := GVL_CONFIG_HISTORY.G_History_Index;
    GVL_CONFIG_HISTORY.G_History_Version[L_Index] := GVL_CONFIG_CONTROL.G_Config_Version;
    GVL_CONFIG_HISTORY.G_History_Time_MS[L_Index] := GVL_TIME_SERVICE.G_Now_MS;
    GVL_CONFIG_HISTORY.G_History_Action[L_Index] := 'APPLY';

    L_Index := L_Index + 1;
    IF L_Index > 5 THEN L_Index := 1; END_IF;
    GVL_CONFIG_HISTORY.G_History_Index := L_Index;

    GVL_CONFIG_CONTROL.G_Backup_Valid := TRUE;
    GVL_CONFIG_CONTROL.G_Apply_Done := TRUE;
END_IF;

GVL_CONFIG_VALIDATION.G_Config_Valid := NOT L_Error;
GVL_CONFIG_VALIDATION.G_Config_Last_Update_MS := GVL_TIME_SERVICE.G_Now_MS;

// >>> BULK_SYNC_ANCHOR: PRG_Config_Manager <<<
          
END_PROGRAM

PROGRAM PRG_Runtime_Budget_Governor

            // RUNTIME BUDGET ENFORCEMENT
// READ-ONLY / NON-INVASIVE

GVL_RUNTIME_BUDGET_ENFORCEMENT.Runtime_Budget_Pressure_Observed :=
    GVL_CANONICAL_RUNTIME_FABRIC_REGISTRY.Runtime_Complexity_Pressure_Observed;

GVL_RUNTIME_BUDGET_ENFORCEMENT.Governance_Runtime_Overhead_Observed :=
    GVL_CANONICAL_RUNTIME_FABRIC_REGISTRY.Governance_Runtime_Cost_Observed;

GVL_RUNTIME_BUDGET_ENFORCEMENT.Verification_Runtime_Budget_Observed :=
    GVL_CANONICAL_RUNTIME_FABRIC_REGISTRY.Verification_Chaining_Limit_Reached;

GVL_RUNTIME_BUDGET_ENFORCEMENT.Observability_Runtime_Budget_Observed :=
    GVL_CANONICAL_RUNTIME_FABRIC_REGISTRY.Observability_Amplification_Limit_Reached;

IF GVL_RUNTIME_BUDGET_ENFORCEMENT.Runtime_Budget_Pressure_Observed THEN
    GVL_RUNTIME_BUDGET_ENFORCEMENT.Runtime_Stability_Budget_At_Risk := TRUE;
END_IF;

IF GVL_RUNTIME_BUDGET_ENFORCEMENT.Verification_Runtime_Budget_Observed THEN
    GVL_RUNTIME_BUDGET_ENFORCEMENT.Verification_Time_Budget_Exceeded := TRUE;
    GVL_RUNTIME_BUDGET_ENFORCEMENT.Verification_Induced_Runtime_Risk := TRUE;
END_IF;

IF GVL_RUNTIME_BUDGET_ENFORCEMENT.Observability_Runtime_Budget_Observed THEN
    GVL_RUNTIME_BUDGET_ENFORCEMENT.Observability_Amplification_Budget_Exceeded := TRUE;
END_IF;
          
END_PROGRAM

PROGRAM PRG_Actuation_Authority_Governor
  VAR
    L_Now_MS : UDINT;
    L_Actuation_Valid : BOOL := TRUE;
    L_Error_Code : UDINT := 0;
    L_Error_Text : STRING(160) := '';
  END_VAR

            L_Now_MS := GVL_STATUS.G_System_Time_MS;
L_Actuation_Valid := TRUE;
L_Error_Code := 0;
L_Error_Text := '';

GVL_ACTUATION_AUTHORITY.Actuation_Authority_Valid := FALSE;
GVL_ACTUATION_AUTHORITY.Actuation_Authority_Granted := FALSE;
GVL_ACTUATION_AUTHORITY.Actuation_Quarantine_Active := TRUE;
GVL_ACTUATION_AUTHORITY.Field_Device_ACK_Valid := FALSE;
GVL_ACTUATION_AUTHORITY.Actuator_Transition_Observed := FALSE;
GVL_ACTUATION_AUTHORITY.Physical_Convergence_Confirmed := FALSE;
GVL_ACTUATION_AUTHORITY.Stable_Physical_Convergence := FALSE;

GVL_ACTUATION_AUTHORITY.Actuation_Command_Epoch := ULINT_TO_UDINT(GVL_OUTPUT_EPOCH.Output_Publication_Epoch);

IF GVL_ACTUATION_AUTHORITY.Field_ACK_Epoch <> GVL_ACTUATION_AUTHORITY.Actuation_Command_Epoch THEN
    GVL_ACTUATION_AUTHORITY.Command_Actuation_Skew_Detected := TRUE;
    L_Actuation_Valid := FALSE;
    L_Error_Code := 26000;
    L_Error_Text := 'Command actuation epoch skew detected';
END_IF;

IF L_Actuation_Valid AND GVL_ACTUATION_AUTHORITY.ACK_Replay_Suspected THEN
    L_Actuation_Valid := FALSE;
    L_Error_Code := 26001;
    L_Error_Text := 'Field ACK replay suspected';
END_IF;

IF L_Actuation_Valid AND GVL_ACTUATION_AUTHORITY.Write_Without_Confirm_Detected THEN
    L_Actuation_Valid := FALSE;
    L_Error_Code := 26002;
    L_Error_Text := 'Write without field confirmation detected';
END_IF;

IF L_Actuation_Valid AND GVL_ACTUATION_AUTHORITY.Relay_Weld_Suspected THEN
    L_Actuation_Valid := FALSE;
    L_Error_Code := 26003;
    L_Error_Text := 'Relay weld suspected';
END_IF;

IF L_Actuation_Valid AND GVL_ACTUATION_AUTHORITY.Actuator_Stall_Detected THEN
    L_Actuation_Valid := FALSE;
    L_Error_Code := 26004;
    L_Error_Text := 'Actuator stall detected';
END_IF;

IF L_Actuation_Valid AND GVL_ACTUATION_AUTHORITY.Partial_Actuation_Detected THEN
    L_Actuation_Valid := FALSE;
    L_Error_Code := 26005;
    L_Error_Text := 'Partial actuation detected';
END_IF;

IF L_Actuation_Valid AND NOT GVL_ACTUATION_AUTHORITY.Current_Signature_Confirmed THEN
    L_Actuation_Valid := FALSE;
    L_Error_Code := 26010;
    L_Error_Text := 'Current signature confirmation missing';
END_IF;

IF L_Actuation_Valid AND NOT GVL_ACTUATION_AUTHORITY.Flow_Response_Confirmed THEN
    L_Actuation_Valid := FALSE;
    L_Error_Code := 26011;
    L_Error_Text := 'Flow response confirmation missing';
END_IF;

IF L_Actuation_Valid AND NOT GVL_ACTUATION_AUTHORITY.Pressure_Response_Confirmed THEN
    L_Actuation_Valid := FALSE;
    L_Error_Code := 26012;
    L_Error_Text := 'Pressure response confirmation missing';
END_IF;

IF L_Actuation_Valid AND NOT GVL_ACTUATION_AUTHORITY.Motion_Response_Confirmed THEN
    L_Actuation_Valid := FALSE;
    L_Error_Code := 26013;
    L_Error_Text := 'Motion response confirmation missing';
END_IF;

IF L_Actuation_Valid THEN
    GVL_ACTUATION_AUTHORITY.Actuation_Authority_Valid := TRUE;
    GVL_ACTUATION_AUTHORITY.Actuation_Authority_Granted := TRUE;
    GVL_ACTUATION_AUTHORITY.Actuation_Quarantine_Active := FALSE;
    GVL_ACTUATION_AUTHORITY.Field_Device_ACK_Valid := TRUE;
    GVL_ACTUATION_AUTHORITY.Actuator_Transition_Observed := TRUE;
    GVL_ACTUATION_AUTHORITY.Physical_Convergence_Confirmed := TRUE;
    GVL_ACTUATION_AUTHORITY.Stable_Physical_Convergence := TRUE;
    GVL_ACTUATION_AUTHORITY.Actuation_Authority_Epoch := GVL_ACTUATION_AUTHORITY.Actuation_Command_Epoch;
    GVL_ACTUATION_AUTHORITY.Actuation_Last_Update_MS := L_Now_MS;
    GVL_ACTUATION_AUTHORITY.Actuation_Lease_Expired := FALSE;
    GVL_ACTUATION_AUTHORITY.Actuation_Last_Error_Code := 0;
    GVL_ACTUATION_AUTHORITY.Actuation_Last_Error_Text := '';
ELSE
    GVL_ACTUATION_AUTHORITY.Actuation_Authority_Valid := FALSE;
    GVL_ACTUATION_AUTHORITY.Actuation_Authority_Granted := FALSE;
    GVL_ACTUATION_AUTHORITY.Actuation_Quarantine_Active := TRUE;
    GVL_ACTUATION_AUTHORITY.Actuation_Lease_Expired := TRUE;
    GVL_ACTUATION_AUTHORITY.Actuation_Last_Error_Code := L_Error_Code;
    GVL_ACTUATION_AUTHORITY.Actuation_Last_Error_Text := L_Error_Text;
    GVL_ACTUATION_AUTHORITY.Actuation_Invalidation_Count := GVL_ACTUATION_AUTHORITY.Actuation_Invalidation_Count + 1;
END_IF;
          
END_PROGRAM

PROGRAM PRG_Water
  VAR
    fbProjection : FB_Water_Output_Projection;
    L_Zone_Enable : ARRAY[1..GVL_CONSTANTS.C_MAX_WATER_ZONES] OF BOOL;
    L_Valve_35_Close : BOOL;
    L_Valve_36_Close : BOOL;
    L_i : INT;
    L_Projected_Valve_Group : UINT;
  END_VAR

            // ==============================================================================
// Water runtime output bridge.
//
// GVL_COMMAND_SHADOW remains owned exclusively by PRG_Command_Arbitration.
// This PRG is the water domain output projection bridge into GVL_WATER_OUTPUT.
//
// Priority:
// 1. Existing global safety close command from command shadow.
// 2. Deterministic water output projection if valid.
//
// This PRG does not perform leak classification, topology decisions,
// diagnostics, or recovery governance.
// ==============================================================================

FOR L_i := 1 TO GVL_CONSTANTS.C_MAX_WATER_ZONES DO
    L_Zone_Enable[L_i] := FALSE;
END_FOR;

IF GVL_INTENT_SAFETY.I_Water_Selective_Recovery_Allowed THEN
    IF (GVL_INTENT_SAFETY.I_Water_Recovery_Target_Zone >= 1) AND (GVL_INTENT_SAFETY.I_Water_Recovery_Target_Zone <= GVL_CONSTANTS.C_MAX_WATER_ZONES) THEN
        L_Zone_Enable[GVL_INTENT_SAFETY.I_Water_Recovery_Target_Zone] := TRUE;
    END_IF;
END_IF;

// Existing authoritative global fallback path.
L_Valve_35_Close := GVL_COMMAND_SHADOW.G_Close_Valve_35;
L_Valve_36_Close := GVL_COMMAND_SHADOW.G_Close_Valve_36;

// Deterministic projection bridge.
// Conservative global fallback projection dominates selective projection.
IF GVL_Water_Output_Projection.G_Runtime_Valid THEN

    IF GVL_Water_Output_Projection.G_Global_Fallback_Projecting THEN
        L_Valve_35_Close := TRUE;
        L_Valve_36_Close := TRUE;
    ELSE
        FOR L_i := 1 TO GVL_CONSTANTS.C_MAX_FLOOD_SENSORS DO
            IF GVL_Water_Output_Projection.G_Output_Projection_State[L_i].Projection_Allowed AND
               GVL_Water_Output_Projection.G_Output_Projection_State[L_i].Physical_Close_Project THEN

                L_Projected_Valve_Group :=
                    GVL_Water_Output_Projection.G_Output_Projection_State[L_i].Valve_Group_Id;

                CASE L_Projected_Valve_Group OF
                    1:
                        L_Valve_35_Close := TRUE;
                    2:
                        L_Valve_36_Close := TRUE;
                    3:
                        L_Valve_35_Close := TRUE;
                        L_Valve_36_Close := TRUE;
                ELSE
                    // Unknown valve group is not projected here.
                    // Conservative fallback is handled by authority/projection layers.
                END_CASE;
            END_IF;
        END_FOR;
    END_IF;
END_IF;

fbProjection(
    VI_Zone_Enable := L_Zone_Enable,
    VI_Valve_35_Close := L_Valve_35_Close,
    VI_Valve_36_Close := L_Valve_36_Close
);

// >>> BULK_SYNC_ANCHOR: PRG_Water <<<
          
END_PROGRAM

PROGRAM PRG_Recovery_Reactivation_Control_Governor

            IF GVL_RECOVERY_ORDERING_INTEGRITY_FABRIC.Recovery_Ordering_Integrity_Valid
AND NOT GVL_RECOVERY_REACTIVATION_CONTROL_FABRIC.Unsafe_Reactivation_Ordering_Detected
AND NOT GVL_RECOVERY_REACTIVATION_CONTROL_FABRIC.Partial_Reactivation_Leak_Detected
AND NOT GVL_RECOVERY_REACTIVATION_CONTROL_FABRIC.CrossSubsystem_Reactivation_Fork THEN

    GVL_RECOVERY_REACTIVATION_CONTROL_FABRIC.Recovery_Reactivation_Control_Valid := TRUE;
    GVL_RECOVERY_REACTIVATION_CONTROL_FABRIC.Recovery_Reactivation_Control_Granted := TRUE;
    GVL_RECOVERY_REACTIVATION_CONTROL_FABRIC.Recovery_Reactivation_Boundary_Stable := TRUE;
    GVL_RECOVERY_REACTIVATION_CONTROL_FABRIC.CrossSubsystem_Reactivation_Consistent := TRUE;
    GVL_RECOVERY_REACTIVATION_CONTROL_FABRIC.Reactivation_Energy_Boundary_Safe := TRUE;
END_IF;
          
END_PROGRAM

PROGRAM PRG_User_Adapt_Control
  VAR
    fbTrace : FB_Trace_Write;
    L_Text : STRING(64);
  END_VAR

            IF GVL_INTENT_USER.I_Set_Adapt_Profile_Req THEN

    // block if safety active
    IF (GVL_SAFETY_SHUTDOWN.G_Safety_Mode <> NORMAL) OR GVL_SAFETY_RECOVERY.G_Recovery_Active THEN

        fbTrace(
            iLayer := TRACE_USER,
            iSource := SRC_USER,
            iReason := REASON_SAFETY,
            iValueBool := FALSE,
            iValueReal := 0.0,
            iText := 'Profile change blocked: SAFETY ACTIVE'
        );

    ELSE

        IF (GVL_INTENT_USER.I_Set_Adapt_Profile_Confirm)
           AND (GVL_INTENT_USER.I_User_Access_Level >= 2) THEN

            GVL_BEHAVIOR_ADAPT.G_Adapt_Profile :=
                GVL_INTENT_USER.I_Adapt_Profile_Value;

            IF GVL_INTENT_USER.I_Adapt_Profile_Value = ADAPT_PROFILE_STABLE THEN
                L_Text := 'Adapt profile: STABLE';
            ELSIF GVL_INTENT_USER.I_Adapt_Profile_Value = ADAPT_PROFILE_BALANCED THEN
                L_Text := 'Adapt profile: BALANCED';
            ELSE
                L_Text := 'Adapt profile: AGGRESSIVE';
            END_IF;

            fbTrace(
                iLayer := TRACE_USER,
                iSource := SRC_USER,
                iReason := REASON_USER_REQUEST,
                iValueBool := TRUE,
                iValueReal := TO_REAL(GVL_INTENT_USER.I_User_Access_Level),
                iText := L_Text
            );

        END_IF;

    END_IF;

    GVL_INTENT_USER.I_Set_Adapt_Profile_Req := FALSE;
    GVL_INTENT_USER.I_Set_Adapt_Profile_Confirm := FALSE;

END_IF;
          
END_PROGRAM

PROGRAM PRG_PreOutput_Safety_Barrier
  VAR
    L_i : INT;
    L_Now_MS : UDINT;
    L_Block_IO : BOOL := FALSE;
    L_Error_Code : UDINT := 0;
    L_Error_Text : STRING(160) := '';
    L_Any_Manifold_Pump_On : BOOL := FALSE;
    L_Prev_Block_IO : BOOL;
    L_Selective_Projection_Active : BOOL;
    L_Global_Fallback_Active : BOOL;
    L_Runtime_Projection_Healthy : BOOL;
    L_Finalized_Publication_Continuity : BOOL;
    L_Physical_Causality_Healthy : BOOL;
    L_Command_Telemetry_Epoch_Aligned : BOOL;
    L_Physical_Ack_Fresh : BOOL;
    fbLog : FB_LogEvent;
  END_VAR

            L_Now_MS := GVL_STATUS.G_System_Time_MS;
L_Block_IO := FALSE;
L_Error_Code := 0;
L_Error_Text := '';
L_Any_Manifold_Pump_On := FALSE;
L_Prev_Block_IO := GVL_COMMAND_VERIFY.PreOutput_Block_IO;

L_Selective_Projection_Active :=
    GVL_Water_Isolation_Authority.G_Any_Selective_Authority_Allowed;

L_Global_Fallback_Active :=
    GVL_Water_Isolation_Authority.G_Any_Global_Fallback_Required;

L_Runtime_Projection_Healthy :=
    GVL_Water_Output_Reconciliation.G_Runtime_Valid
    AND NOT GVL_Water_Output_Reconciliation.G_Any_Conflict_Detected;

// Command ↔ telemetry epoch binding.
L_Command_Telemetry_Epoch_Aligned :=
    GVL_TELEMETRY.Command_Epoch = GVL_OUTPUT_EPOCH.Output_Publication_Epoch
    AND GVL_TELEMETRY.Telemetry_Epoch = GVL_OUTPUT_EPOCH.Output_Publication_Epoch
    AND GVL_TELEMETRY.Telemetry_Epoch >=
        GVL_TELEMETRY.Last_Acknowledged_Command_Epoch;

// Physical acknowledgment freshness.
L_Physical_Ack_Fresh :=
    (L_Now_MS - GVL_TELEMETRY.Last_Physical_Ack_Time_MS) <= 5000;

// Physical causality evidence.
L_Physical_Causality_Healthy :=
    GVL_TELEMETRY.Telemetry_Runtime_Valid
    AND GVL_TELEMETRY.Telemetry_Freshness_Valid
    AND NOT GVL_TELEMETRY.Telemetry_Lease_Expired
    AND NOT GVL_TELEMETRY.Telemetry_Quarantine_Active
    AND GVL_TELEMETRY.Command_Telemetry_Causality_Valid
    AND NOT GVL_TELEMETRY.Command_Telemetry_Divergence_Detected
    AND GVL_TELEMETRY.Actuator_Feedback_Valid
    AND GVL_TELEMETRY.Actuator_Feedback_Fresh
    AND GVL_TELEMETRY.Physical_Effect_Confirmed
    AND L_Command_Telemetry_Epoch_Aligned
    AND L_Physical_Ack_Fresh
    AND NOT GVL_TELEMETRY.Telemetry_Replay_Suspected;

// Finalized publication continuity proof chain.
L_Finalized_Publication_Continuity :=
    GVL_SEMANTIC_PROGRESS.Semantic_Forward_Progress_Valid
    AND GVL_SEMANTIC_PROGRESS.Semantic_Execution_Continuity_OK
    AND NOT GVL_SEMANTIC_PROGRESS.Semantic_Stagnation_Detected
    AND NOT GVL_SEMANTIC_PROGRESS.Semantic_Replay_Suspected
    AND NOT GVL_SEMANTIC_PROGRESS.Semantic_Livelock_Suspected
    AND NOT GVL_SEMANTIC_PROGRESS.Semantic_Deadlock_Suspected
    AND NOT GVL_SEMANTIC_PROGRESS.Semantic_Progress_Lease_Expired
    AND NOT GVL_SEMANTIC_PROGRESS.Semantic_Progress_Quarantine_Active
    AND GVL_RUNTIME_SNAPSHOT.Snapshot_Frozen
    AND GVL_RUNTIME_SNAPSHOT.Snapshot_Publication_Allowed
    AND GVL_RUNTIME_SNAPSHOT.Snapshot_Copy_Valid
    AND GVL_RUNTIME_SNAPSHOT.Snapshot_Isolation_Valid
    AND NOT GVL_RUNTIME_SNAPSHOT.Snapshot_Mutation_Detected
    AND GVL_DISTRIBUTED_SNAPSHOT.Distributed_Publication_Reconciled
    AND GVL_DISTRIBUTED_SNAPSHOT.Distributed_Publication_Freeze_Valid
    AND GVL_DISTRIBUTED_SNAPSHOT.Distributed_Snapshot_Consistent
    AND GVL_DISTRIBUTED_COMMIT.Distributed_Commit_Valid
    AND GVL_DISTRIBUTED_COMMIT.Publication_Prepare_Valid
    AND GVL_DISTRIBUTED_COMMIT.Publication_Commit_Confirmed
    AND NOT GVL_DISTRIBUTED_COMMIT.Peer_Commit_Mismatch
    AND NOT GVL_DISTRIBUTED_COMMIT.Distributed_Commit_Quarantine_Active
    AND NOT GVL_DISTRIBUTED_COMMIT.Commit_Lease_Expired
    AND GVL_OUTPUT_EPOCH.Output_Publication_Valid
    AND GVL_OUTPUT_EPOCH.Output_Runtime_Epoch_Valid
    AND NOT GVL_OUTPUT_EPOCH.Output_Lease_Expired
    AND NOT GVL_OUTPUT_EPOCH.Output_Forced_Safe_Decay;

IF (NOT L_Block_IO)
   AND (NOT L_Finalized_Publication_Continuity) THEN
    L_Block_IO := TRUE;
    L_Error_Code := 3999;
    L_Error_Text := 'PreOutput finalized publication continuity invalid';
END_IF;

IF (NOT L_Block_IO)
   AND (NOT L_Physical_Causality_Healthy) THEN
    L_Block_IO := TRUE;
    L_Error_Code := 3998;
    L_Error_Text := 'Physical causality evidence invalid';
END_IF;

IF (NOT L_Block_IO) AND (NOT GVL_STATUS.G_Is_Active_PLC) THEN
    L_Block_IO := TRUE;
    L_Error_Code := 4000;
    L_Error_Text := 'PreOutput inactive PLC';
END_IF;

IF (NOT L_Block_IO)
   AND (GVL_COMMAND.G_Gas_Valve_Close <> GVL_COMMAND_SHADOW.G_Gas_Valve_Close) THEN
    L_Block_IO := TRUE;
    L_Error_Code := 4001;
    L_Error_Text := 'PreOutput gas command mismatch';
END_IF;

IF (NOT L_Block_IO)
   AND (GVL_COMMAND.G_Boiler_Stop <> GVL_COMMAND_SHADOW.G_Boiler_Stop) THEN
    L_Block_IO := TRUE;
    L_Error_Code := 4002;
    L_Error_Text := 'PreOutput boiler command mismatch';
END_IF;

IF (NOT L_Block_IO)
   AND (GVL_COMMAND.G_Vent_Stop <> GVL_COMMAND_SHADOW.G_Vent_Stop) THEN
    L_Block_IO := TRUE;
    L_Error_Code := 4003;
    L_Error_Text := 'PreOutput vent command mismatch';
END_IF;

IF (NOT L_Block_IO)
   AND (GVL_COMMAND.G_Close_Valve_35 <> GVL_COMMAND_SHADOW.G_Close_Valve_35) THEN
    L_Block_IO := TRUE;
    L_Error_Code := 4004;
    L_Error_Text := 'PreOutput valve 35 command mismatch';
END_IF;

IF (NOT L_Block_IO)
   AND (GVL_COMMAND.G_Close_Valve_36 <> GVL_COMMAND_SHADOW.G_Close_Valve_36) THEN
    L_Block_IO := TRUE;
    L_Error_Code := 4005;
    L_Error_Text := 'PreOutput valve 36 command mismatch';
END_IF;

GVL_COMMAND_VERIFY.PreOutput_Physical_Causality_Valid :=
    L_Physical_Causality_Healthy;

GVL_COMMAND_VERIFY.PreOutput_Barrier_OK := NOT L_Block_IO;
GVL_COMMAND_VERIFY.PreOutput_Block_IO := L_Block_IO;
GVL_COMMAND_VERIFY.PreOutput_Last_Error_Code := L_Error_Code;
GVL_COMMAND_VERIFY.PreOutput_Last_Error_Text := L_Error_Text;

IF L_Block_IO THEN
    GVL_COMMAND_VERIFY.PreOutput_Last_Error_Time_MS := L_Now_MS;
    IF NOT L_Prev_Block_IO THEN
        GVL_COMMAND_VERIFY.PreOutput_Block_Count :=
            GVL_COMMAND_VERIFY.PreOutput_Block_Count + 1;
        fbLog(
            VI_Event_Type := 1002,
            VI_Timestamp := L_Now_MS,
            VI_Param1 := L_Error_Code,
            VI_Param2 := GVL_COMMAND_VERIFY.PreOutput_Block_Count
        );
    END_IF;
END_IF;
          
END_PROGRAM

PROGRAM PRG_Runtime_Transition_Validator

            // PASSIVE FORMAL TRANSITION VALIDATOR
// NO EXECUTION MUTATION
// NO AUTHORITY MUTATION
// OBSERVABILITY ONLY

GVL_RUNTIME_TRANSITION_SYSTEM.Runtime_Transition_Legal := FALSE;
GVL_RUNTIME_TRANSITION_SYSTEM.Runtime_Transition_Proofs_Valid := FALSE;
GVL_RUNTIME_TRANSITION_SYSTEM.Runtime_Transition_Lineage_Valid := FALSE;
GVL_RUNTIME_TRANSITION_SYSTEM.Runtime_Transition_Temporal_Valid := FALSE;

CASE GVL_RUNTIME_STATE_ALGEBRA.Current_Runtime_State OF

    SYS_SAFE:
        GVL_RUNTIME_TRANSITION_SYSTEM.Runtime_Transition_Legal := TRUE;
        GVL_RUNTIME_TRANSITION_SYSTEM.Runtime_Transition_Proofs_Valid := TRUE;

    SYS_RECOVERING:
        GVL_RUNTIME_TRANSITION_SYSTEM.Runtime_Transition_Legal :=
            GVL_TEMPORAL_CAUSALITY_CLOSURE_FABRIC.Temporal_Causality_Coherent;

        GVL_RUNTIME_TRANSITION_SYSTEM.Runtime_Transition_Proofs_Valid :=
            GVL_SAFETY_OBSERVABILITY_TRUTH_FABRIC.Observability_Reality_Equivalence_Granted;

        GVL_RUNTIME_TRANSITION_SYSTEM.Runtime_Transition_Lineage_Valid :=
            GVL_AUTHORITY_LINEAGE.Authority_Lineage_Valid;

        GVL_RUNTIME_TRANSITION_SYSTEM.Runtime_Transition_Temporal_Valid :=
            GVL_DISTRIBUTED_EPOCH_LINEARITY_FABRIC.Epoch_Timeline_Monotonic;

    SYS_QUARANTINED:
        GVL_RUNTIME_TRANSITION_SYSTEM.Runtime_Transition_Legal := TRUE;

    SYS_TRUSTLESS:
        GVL_RUNTIME_TRANSITION_SYSTEM.Runtime_Transition_Legal := FALSE;
        GVL_RUNTIME_TRANSITION_SYSTEM.Unsafe_Trust_Escalation_Observed := TRUE;

ELSE
    GVL_RUNTIME_TRANSITION_SYSTEM.Illegal_Runtime_Transition_Observed := TRUE;

END_CASE;
          
END_PROGRAM

PROGRAM PRG_Power_Domain_Segmentation_Governor

            IF GVL_RESIDUAL_ENERGY_STATE_FABRIC.Residual_Energy_State_Valid
AND NOT GVL_POWER_DOMAIN_SEGMENTATION_FABRIC.Unsafe_Power_Resurrection_Detected
AND NOT GVL_POWER_DOMAIN_SEGMENTATION_FABRIC.Partial_Power_Isolation_Asymmetry
AND NOT GVL_POWER_DOMAIN_SEGMENTATION_FABRIC.Distributed_Power_Segmentation_Fork THEN

    GVL_POWER_DOMAIN_SEGMENTATION_FABRIC.Power_Domain_Segmentation_Valid := TRUE;
    GVL_POWER_DOMAIN_SEGMENTATION_FABRIC.Power_Domain_Segmentation_Granted := TRUE;
    GVL_POWER_DOMAIN_SEGMENTATION_FABRIC.Power_Domain_Boundaries_Canonical := TRUE;
    GVL_POWER_DOMAIN_SEGMENTATION_FABRIC.Distributed_Power_Segmentation_Stable := TRUE;
    GVL_POWER_DOMAIN_SEGMENTATION_FABRIC.Power_Reactivation_Isolation_Valid := TRUE;
END_IF;
          
END_PROGRAM

PROGRAM PRG_OpenTherm_Adapter_Status
  VAR
    L_i : INT;
    L_Now_MS : UDINT;
    L_Heartbeat_Age : UDINT;
    L_Command_Age : UDINT;
  END_VAR

            L_Now_MS := GVL_STATUS.G_System_Time_MS;

FOR L_i := 1 TO GVL_CONSTANTS.C_MAX_BOILERS DO

    // ======================================================
    // HEARTBEAT VALIDATION
    // ======================================================
    IF GVL_OPENTHERM_ADAPTER.G_Status[L_i].Raw_Heartbeat <>
       GVL_OPENTHERM_ADAPTER.G_Status[L_i].Last_Heartbeat THEN

        GVL_OPENTHERM_ADAPTER.G_Status[L_i].Last_Heartbeat :=
            GVL_OPENTHERM_ADAPTER.G_Status[L_i].Raw_Heartbeat;

        GVL_OPENTHERM_ADAPTER.G_Status[L_i].Last_Heartbeat_MS := L_Now_MS;
    END_IF;

    L_Heartbeat_Age :=
        L_Now_MS - GVL_OPENTHERM_ADAPTER.G_Status[L_i].Last_Heartbeat_MS;

    GVL_OPENTHERM_ADAPTER.G_Status[L_i].Heartbeat_Age_MS :=
        L_Heartbeat_Age;

    GVL_OPENTHERM_ADAPTER.G_Status[L_i].Heartbeat_Timeout :=
        (L_Heartbeat_Age > GVL_CONFIG.G_OpenTherm_Heartbeat_Timeout_MS);

    // ======================================================
    // COMMAND ACK VALIDATION
    // ======================================================
    GVL_OPENTHERM_ADAPTER.G_Status[L_i].Command_Ack :=
        (GVL_OPENTHERM_ADAPTER.G_Status[L_i].Raw_Ack_Seq =
         GVL_OPENTHERM_ADAPTER.G_Command[L_i].Sequence);

    GVL_OPENTHERM_ADAPTER.G_Status[L_i].Last_Command_Ack_Seq :=
        GVL_OPENTHERM_ADAPTER.G_Status[L_i].Raw_Ack_Seq;

    L_Command_Age :=
        L_Now_MS - GVL_OPENTHERM_ADAPTER.G_Command[L_i].Last_Write_MS;

    GVL_OPENTHERM_ADAPTER.G_Status[L_i].Command_Age_MS :=
        L_Command_Age;

    GVL_OPENTHERM_ADAPTER.G_Status[L_i].Command_Timeout :=
        (NOT GVL_OPENTHERM_ADAPTER.G_Status[L_i].Command_Ack) AND
        (L_Command_Age > GVL_CONFIG.G_OpenTherm_Command_Ack_Timeout_MS);

    // ======================================================
    // FINAL ADAPTER STATE
    // ======================================================
    GVL_OPENTHERM_ADAPTER.G_Status[L_i].Adapter_Online :=
        GVL_OPENTHERM_ADAPTER.G_Status[L_i].Raw_Online AND
        (NOT GVL_OPENTHERM_ADAPTER.G_Status[L_i].Heartbeat_Timeout) AND
        (NOT GVL_OPENTHERM_ADAPTER.G_Status[L_i].Command_Timeout);

    GVL_OPENTHERM_ADAPTER.G_Status[L_i].Adapter_Error :=
        GVL_OPENTHERM_ADAPTER.G_Status[L_i].Raw_Error OR
        GVL_OPENTHERM_ADAPTER.G_Status[L_i].Command_Timeout OR
        GVL_OPENTHERM_ADAPTER.G_Status[L_i].Heartbeat_Timeout;

    // ======================================================
    // ENUM STATES
    // ======================================================
    IF GVL_OPENTHERM_ADAPTER.G_Status[L_i].Heartbeat_Timeout THEN
        GVL_OPENTHERM_ADAPTER.G_Status[L_i].Adapter_State := OT_STATE_HEARTBEAT_TIMEOUT;
        GVL_OPENTHERM_ADAPTER.G_Status[L_i].Error_State := OT_ERROR_HEARTBEAT_TIMEOUT;

    ELSIF GVL_OPENTHERM_ADAPTER.G_Status[L_i].Command_Timeout THEN
        GVL_OPENTHERM_ADAPTER.G_Status[L_i].Adapter_State := OT_STATE_ACK_TIMEOUT;
        GVL_OPENTHERM_ADAPTER.G_Status[L_i].Error_State := OT_ERROR_ACK_TIMEOUT;

    ELSIF GVL_OPENTHERM_ADAPTER.G_Status[L_i].Raw_Error THEN
        GVL_OPENTHERM_ADAPTER.G_Status[L_i].Adapter_State := OT_STATE_ADAPTER_ERROR;
        GVL_OPENTHERM_ADAPTER.G_Status[L_i].Error_State := OT_ERROR_ADAPTER_FAULT;

    ELSIF GVL_OPENTHERM_ADAPTER.G_Status[L_i].Adapter_Online THEN
        GVL_OPENTHERM_ADAPTER.G_Status[L_i].Adapter_State := OT_STATE_ONLINE;
        GVL_OPENTHERM_ADAPTER.G_Status[L_i].Error_State := OT_ERROR_NONE;

    ELSE
        GVL_OPENTHERM_ADAPTER.G_Status[L_i].Adapter_State := OT_STATE_OFFLINE;
        GVL_OPENTHERM_ADAPTER.G_Status[L_i].Error_State := OT_ERROR_COMMUNICATION;
    END_IF;

    // ======================================================
    // PUBLISH TO SYSTEM STATE
    // ======================================================
    GVL_STATE.G_Boiler_OT_Online[L_i] :=
        GVL_OPENTHERM_ADAPTER.G_Status[L_i].Adapter_Online;

    GVL_STATE.G_Boiler_OT_Command_Ack[L_i] :=
        GVL_OPENTHERM_ADAPTER.G_Status[L_i].Command_Ack;

    GVL_STATE.G_Boiler_OT_Command_Timeout[L_i] :=
        GVL_OPENTHERM_ADAPTER.G_Status[L_i].Command_Timeout;

    GVL_STATE.G_Boiler_OT_Heartbeat_Timeout[L_i] :=
        GVL_OPENTHERM_ADAPTER.G_Status[L_i].Heartbeat_Timeout;

    GVL_STATE.G_Boiler_OT_Adapter_Error[L_i] :=
        GVL_OPENTHERM_ADAPTER.G_Status[L_i].Adapter_Error;

    GVL_STATE.G_Boiler_OT_Heartbeat_Age_MS[L_i] :=
        GVL_OPENTHERM_ADAPTER.G_Status[L_i].Heartbeat_Age_MS;

    GVL_STATE.G_Boiler_OT_Command_Age_MS[L_i] :=
        GVL_OPENTHERM_ADAPTER.G_Status[L_i].Command_Age_MS;

    GVL_STATE.G_Boiler_OT_Adapter_State[L_i] :=
        GVL_OPENTHERM_ADAPTER.G_Status[L_i].Adapter_State;

    GVL_STATE.G_Boiler_OT_Error_State[L_i] :=
        GVL_OPENTHERM_ADAPTER.G_Status[L_i].Error_State;

    GVL_STATE.G_Boiler_Error[L_i] :=
        GVL_OPENTHERM_ADAPTER.G_Status[L_i].Adapter_Error;

    GVL_STATE.G_Boiler_Flame[L_i] :=
        GVL_OPENTHERM_ADAPTER.G_Status[L_i].Raw_Flame;

END_FOR;
          
END_PROGRAM

PROGRAM PRG_Proof_Continuity_Audit_Governor

            // PASSIVE PROOF AUDIT ONLY

GVL_PROOF_CONTINUITY_AUDIT_FABRIC.Proof_Continuity_Observed :=
    GVL_SEMANTIC_DRIFT_OBSERVABILITY_FABRIC.Semantic_Continuity_Observed;

GVL_PROOF_CONTINUITY_AUDIT_FABRIC.Proof_Lineage_Coherent := TRUE;
GVL_PROOF_CONTINUITY_AUDIT_FABRIC.Proof_Historical_Integrity_Observed := TRUE;
          
END_PROGRAM

PROGRAM PRG_Command_Arbitration
  VAR
    L_Mode : E_Safety_Mode;
    L_Safety_Active : BOOL;
    L_User_Access_OK : BOOL;
    L_i : INT;
    L_Gas_Valve_Close : BOOL;
    L_Boiler_Stop : BOOL;
    L_Supply_100_Req : BOOL;
    L_Supply_80_Req : BOOL;
    L_Vent_PV3_Boost : BOOL;
    L_Exhaust_100_Req : BOOL;
    L_Vent_Stop : BOOL;
    L_Vent_Block : BOOL;
    L_Vent_Smoke_Exhaust : BOOL;
    L_Heating_Block : BOOL;
    L_Heating_Emergency_Stop : BOOL;
    L_Heating_Gas_Safety_Stop : BOOL;
    L_Water_Block : BOOL;
    L_Water_Emergency_Stop : BOOL;
    L_Close_Valve_35 : BOOL;
    L_Close_Valve_36 : BOOL;
    L_Lock_1_Open : BOOL;
    L_Lock_1_Close : BOOL;
    L_Lock_2_Open : BOOL;
    L_Lock_2_Close : BOOL;
    L_Gate_Open : BOOL;
    L_Wicket_Open : BOOL;
  END_VAR

            // ======================================================
// PRIORITY 1: PLC ROLE VALIDATION (ABSOLUTE)
// ======================================================
IF GVL_STATUS.G_Is_Active_PLC AND GVL_STATUS.G_Other_PLC_Is_Active THEN
    GVL_HEALTH_BRIDGE.G_Role_Conflict_Error := TRUE;

    GVL_COMMAND_SHADOW.G_Gas_Valve_Close := TRUE;
    GVL_COMMAND_SHADOW.G_Boiler_Stop := TRUE;
    GVL_COMMAND_SHADOW.G_Supply_100_Req := FALSE;
    GVL_COMMAND_SHADOW.G_Supply_80_Req := FALSE;
    GVL_COMMAND_SHADOW.G_Vent_PV3_Boost := FALSE;
    GVL_COMMAND_SHADOW.G_Exhaust_100_Req := FALSE;
    GVL_COMMAND_SHADOW.G_Vent_Stop := TRUE;
    GVL_COMMAND_SHADOW.G_Vent_Block := TRUE;
    GVL_COMMAND_SHADOW.G_Vent_Smoke_Exhaust := FALSE;

    GVL_COMMAND_SHADOW.G_Heating_Block := TRUE;
    GVL_COMMAND_SHADOW.G_Heating_Emergency_Stop := TRUE;
    GVL_COMMAND_SHADOW.G_Heating_Gas_Safety_Stop := TRUE;

    GVL_COMMAND_SHADOW.G_Water_Block := TRUE;
    GVL_COMMAND_SHADOW.G_Water_Emergency_Stop := TRUE;
    GVL_COMMAND_SHADOW.G_Close_Valve_35 := TRUE;
    GVL_COMMAND_SHADOW.G_Close_Valve_36 := TRUE;

    GVL_COMMAND_SHADOW.G_Lock_1_Open := FALSE;
    GVL_COMMAND_SHADOW.G_Lock_1_Close := FALSE;
    GVL_COMMAND_SHADOW.G_Lock_2_Open := FALSE;
    GVL_COMMAND_SHADOW.G_Lock_2_Close := FALSE;
    GVL_COMMAND_SHADOW.G_Gate_Open := FALSE;
    GVL_COMMAND_SHADOW.G_Wicket_Open := FALSE;
    RETURN;
END_IF;

// ======================================================
// PRIORITY 2: PLC INACTIVE
// ======================================================
IF NOT GVL_STATUS.G_Is_Active_PLC THEN
    GVL_COMMAND_SHADOW.G_Gas_Valve_Close := GVL_COMMAND_POLICY_CONFIG.G_PLC_Inactive_Close_Gas;
    GVL_COMMAND_SHADOW.G_Boiler_Stop := GVL_COMMAND_POLICY_CONFIG.G_PLC_Inactive_Stop_Boiler;
    GVL_COMMAND_SHADOW.G_Supply_100_Req := FALSE;
    GVL_COMMAND_SHADOW.G_Supply_80_Req := FALSE;
    GVL_COMMAND_SHADOW.G_Vent_PV3_Boost := FALSE;
    GVL_COMMAND_SHADOW.G_Exhaust_100_Req := FALSE;
    GVL_COMMAND_SHADOW.G_Vent_Stop := GVL_COMMAND_POLICY_CONFIG.G_PLC_Inactive_Stop_Vent;
    GVL_COMMAND_SHADOW.G_Vent_Block := FALSE;
    GVL_COMMAND_SHADOW.G_Vent_Smoke_Exhaust := FALSE;

    GVL_COMMAND_SHADOW.G_Heating_Block := GVL_COMMAND_POLICY_CONFIG.G_PLC_Inactive_Block_Heating;
    GVL_COMMAND_SHADOW.G_Heating_Emergency_Stop := FALSE;
    GVL_COMMAND_SHADOW.G_Heating_Gas_Safety_Stop := FALSE;

    GVL_COMMAND_SHADOW.G_Water_Block := GVL_COMMAND_POLICY_CONFIG.G_PLC_Inactive_Block_Water;
    GVL_COMMAND_SHADOW.G_Water_Emergency_Stop := FALSE;
    GVL_COMMAND_SHADOW.G_Close_Valve_35 := FALSE;
    GVL_COMMAND_SHADOW.G_Close_Valve_36 := FALSE;

    GVL_COMMAND_SHADOW.G_Lock_1_Open := FALSE;
    GVL_COMMAND_SHADOW.G_Lock_1_Close := FALSE;
    GVL_COMMAND_SHADOW.G_Lock_2_Open := FALSE;
    GVL_COMMAND_SHADOW.G_Lock_2_Close := FALSE;
    GVL_COMMAND_SHADOW.G_Gate_Open := FALSE;
    GVL_COMMAND_SHADOW.G_Wicket_Open := FALSE;
    RETURN;
END_IF;

// ======================================================
// RESET LOCAL BUFFER
// ======================================================
L_Gas_Valve_Close := FALSE;
L_Boiler_Stop := FALSE;
L_Supply_100_Req := FALSE;
L_Supply_80_Req := FALSE;
L_Vent_PV3_Boost := FALSE;
L_Exhaust_100_Req := FALSE;
L_Vent_Stop := FALSE;
L_Vent_Block := FALSE;
L_Vent_Smoke_Exhaust := FALSE;

L_Heating_Block := FALSE;
L_Heating_Emergency_Stop := FALSE;
L_Heating_Gas_Safety_Stop := FALSE;

L_Water_Block := FALSE;
L_Water_Emergency_Stop := FALSE;
L_Close_Valve_35 := FALSE;
L_Close_Valve_36 := FALSE;

L_Lock_1_Open := FALSE;
L_Lock_1_Close := FALSE;
L_Lock_2_Open := FALSE;
L_Lock_2_Close := FALSE;
L_Gate_Open := FALSE;
L_Wicket_Open := FALSE;

// ======================================================
// PRIORITY 3: SAFETY MODE
// ======================================================
L_Mode := GVL_SAFETY_SHUTDOWN.G_Safety_Mode;
L_Safety_Active := FALSE;

CASE L_Mode OF

    NORMAL:
        L_Safety_Active := FALSE;

    FIRE:
        L_Safety_Active := TRUE;
        L_Heating_Block := GVL_COMMAND_POLICY_CONFIG.G_Fire_Block_Heating;
        L_Boiler_Stop := GVL_COMMAND_POLICY_CONFIG.G_Fire_Stop_Boiler;
        L_Vent_Stop := FALSE;
        L_Vent_PV3_Boost := FALSE;
        L_Exhaust_100_Req := FALSE;
        L_Vent_Smoke_Exhaust := TRUE;
        L_Heating_Emergency_Stop := GVL_COMMAND_POLICY_CONFIG.G_Fire_Block_Heating;
        L_Lock_1_Open := GVL_COMMAND_POLICY_CONFIG.G_Fire_Open_Lock_1;
        L_Lock_2_Open := GVL_COMMAND_POLICY_CONFIG.G_Fire_Open_Lock_2;
        L_Gate_Open := GVL_COMMAND_POLICY_CONFIG.G_Fire_Open_Gate;
        L_Wicket_Open := GVL_COMMAND_POLICY_CONFIG.G_Fire_Open_Wicket;

    GAS:
        L_Safety_Active := TRUE;
        L_Gas_Valve_Close := GVL_COMMAND_POLICY_CONFIG.G_Gas_Close_Gas;
        L_Boiler_Stop := GVL_COMMAND_POLICY_CONFIG.G_Gas_Stop_Boiler;
        L_Heating_Block := GVL_COMMAND_POLICY_CONFIG.G_Gas_Block_Heating;
        L_Heating_Gas_Safety_Stop := GVL_COMMAND_POLICY_CONFIG.G_Gas_Block_Heating;
        L_Vent_PV3_Boost := TRUE;
        L_Vent_Smoke_Exhaust := FALSE;
        L_Gate_Open := GVL_COMMAND_POLICY_CONFIG.G_Gas_Open_Gate;
        L_Wicket_Open := GVL_COMMAND_POLICY_CONFIG.G_Gas_Open_Wicket;
        L_Lock_1_Open := GVL_COMMAND_POLICY_CONFIG.G_Gas_Open_Lock_1;
        L_Lock_2_Open := GVL_COMMAND_POLICY_CONFIG.G_Gas_Open_Lock_2;

    WATER_LEAK:
        L_Safety_Active := TRUE;
        L_Water_Block := GVL_COMMAND_POLICY_CONFIG.G_Water_Block_Water;
        L_Water_Emergency_Stop := GVL_COMMAND_POLICY_CONFIG.G_Water_Block_Water;
        L_Close_Valve_35 := GVL_COMMAND_POLICY_CONFIG.G_Water_Block_Water;
        L_Close_Valve_36 := GVL_COMMAND_POLICY_CONFIG.G_Water_Block_Water;

    GLOBAL_STOP:
        L_Safety_Active := TRUE;
        L_Heating_Block := GVL_COMMAND_POLICY_CONFIG.G_GlobalStop_Block_Heating;
        L_Heating_Emergency_Stop := GVL_COMMAND_POLICY_CONFIG.G_GlobalStop_Block_Heating;
        L_Boiler_Stop := GVL_COMMAND_POLICY_CONFIG.G_GlobalStop_Stop_Boiler;
        L_Vent_Stop := GVL_COMMAND_POLICY_CONFIG.G_GlobalStop_Stop_Vent;
        L_Water_Block := GVL_COMMAND_POLICY_CONFIG.G_GlobalStop_Block_Water;
        L_Water_Emergency_Stop := GVL_COMMAND_POLICY_CONFIG.G_GlobalStop_Block_Water;
        L_Close_Valve_35 := GVL_COMMAND_POLICY_CONFIG.G_GlobalStop_Block_Water;
        L_Close_Valve_36 := GVL_COMMAND_POLICY_CONFIG.G_GlobalStop_Block_Water;

ELSE
        L_Safety_Active := TRUE;
        L_Gas_Valve_Close := TRUE;
        L_Boiler_Stop := TRUE;
        L_Heating_Block := TRUE;
        L_Heating_Emergency_Stop := TRUE;
        L_Vent_Stop := TRUE;
        L_Water_Block := TRUE;
        L_Water_Emergency_Stop := TRUE;
        L_Close_Valve_35 := TRUE;
        L_Close_Valve_36 := TRUE;
END_CASE;

// ======================================================
// PRIORITY 4: USER INTENT (ONLY WHEN SAFETY IS NOT ACTIVE)
// ======================================================
L_User_Access_OK := GVL_INTENT_USER.I_Source_Valid AND (GVL_INTENT_USER.I_User_Access_Level >= 1);

IF (NOT L_Safety_Active) AND L_User_Access_OK THEN
    IF GVL_INTENT_USER.I_Lock_1_Open_Request THEN
        L_Lock_1_Open := TRUE;
        L_Lock_1_Close := FALSE;
    ELSIF GVL_INTENT_USER.I_Lock_1_Close_Request THEN
        L_Lock_1_Open := FALSE;
        L_Lock_1_Close := TRUE;
    END_IF;

    IF GVL_INTENT_USER.I_Lock_2_Open_Request THEN
        L_Lock_2_Open := TRUE;
        L_Lock_2_Close := FALSE;
    ELSIF GVL_INTENT_USER.I_Lock_2_Close_Request THEN
        L_Lock_2_Open := FALSE;
        L_Lock_2_Close := TRUE;
    END_IF;

    IF GVL_INTENT_USER.I_Gate_Open_Request THEN
        L_Gate_Open := TRUE;
    END_IF;

    IF GVL_INTENT_USER.I_Wicket_Open_Request THEN
        L_Wicket_Open := TRUE;
    END_IF;
END_IF;

// Dangerous user actions require explicit confirmation and elevated access.
IF (NOT L_Safety_Active) AND
   GVL_INTENT_USER.I_Source_Valid AND
   GVL_INTENT_USER.I_Dangerous_Action_Request AND
   GVL_INTENT_USER.I_Dangerous_Action_Confirm AND
   (GVL_INTENT_USER.I_User_Access_Level >= 2) THEN
    // Reserved for future high-risk manual actions.
    // No direct safety override is allowed here.
END_IF;

// ======================================================
// PRIORITY 5: AUTOMATION RULES (ONLY SAFE COMMAND-LEVEL ACTIONS)
// ======================================================
IF NOT L_Safety_Active THEN
    FOR L_i := 1 TO GVL_CONSTANTS.C_MAX_RULES DO
        IF GVL_STATE.G_Rule_Actions[L_i].Active AND GVL_STATE.G_Rule_Actions[L_i].Triggered THEN
            CASE GVL_STATE.G_Rule_Actions[L_i].Action_Type OF

                ACTION_SET_FLOOR_HEATING:
                    IF GVL_STATE.G_Rule_Actions[L_i].Value <= 0.0 THEN
                        L_Heating_Block := TRUE;
                        L_Boiler_Stop := TRUE;
                    END_IF;

                ACTION_SET_VENTILATION:
                    IF GVL_STATE.G_Rule_Actions[L_i].Value <= 0.0 THEN
                        L_Vent_Stop := TRUE;
                    END_IF;

            ELSE
                // Non command-level actions are handled by their own subsystem.
            END_CASE;
        END_IF;
    END_FOR;
END_IF;

// ======================================================
// POST-PROCESS CONFLICT RESOLUTION
// ======================================================
IF (L_Mode = FIRE) AND GVL_COMMAND_POLICY_CONFIG.G_Fire_Block_Lock_Close THEN
    L_Lock_1_Close := FALSE;
    L_Lock_2_Close := FALSE;
END_IF;

IF GVL_COMMAND_POLICY_CONFIG.G_Block_Close_When_Open_Commanded THEN
    IF L_Lock_1_Open AND L_Lock_1_Close THEN
        L_Lock_1_Close := FALSE;
    END_IF;

    IF L_Lock_2_Open AND L_Lock_2_Close THEN
        L_Lock_2_Close := FALSE;
    END_IF;
END_IF;

// ======================================================
// SINGLE POINT WRITE (DETERMINISTIC)
// ======================================================
GVL_COMMAND_SHADOW.G_Gas_Valve_Close := L_Gas_Valve_Close;
GVL_COMMAND_SHADOW.G_Boiler_Stop := L_Boiler_Stop;
GVL_COMMAND_SHADOW.G_Supply_100_Req := L_Supply_100_Req;
GVL_COMMAND_SHADOW.G_Supply_80_Req := L_Supply_80_Req;
GVL_COMMAND_SHADOW.G_Vent_PV3_Boost := L_Vent_PV3_Boost;
GVL_COMMAND_SHADOW.G_Exhaust_100_Req := L_Exhaust_100_Req;
GVL_COMMAND_SHADOW.G_Vent_Stop := L_Vent_Stop;
GVL_COMMAND_SHADOW.G_Vent_Block := L_Vent_Block;
GVL_COMMAND_SHADOW.G_Vent_Smoke_Exhaust := L_Vent_Smoke_Exhaust;

GVL_COMMAND_SHADOW.G_Heating_Block := L_Heating_Block;
GVL_COMMAND_SHADOW.G_Heating_Emergency_Stop := L_Heating_Emergency_Stop;
GVL_COMMAND_SHADOW.G_Heating_Gas_Safety_Stop := L_Heating_Gas_Safety_Stop;

GVL_COMMAND_SHADOW.G_Water_Block := L_Water_Block;
GVL_COMMAND_SHADOW.G_Water_Emergency_Stop := L_Water_Emergency_Stop;
GVL_COMMAND_SHADOW.G_Close_Valve_35 := L_Close_Valve_35;
GVL_COMMAND_SHADOW.G_Close_Valve_36 := L_Close_Valve_36;

GVL_COMMAND_SHADOW.G_Lock_1_Open := L_Lock_1_Open;
GVL_COMMAND_SHADOW.G_Lock_1_Close := L_Lock_1_Close;
GVL_COMMAND_SHADOW.G_Lock_2_Open := L_Lock_2_Open;
GVL_COMMAND_SHADOW.G_Lock_2_Close := L_Lock_2_Close;
GVL_COMMAND_SHADOW.G_Gate_Open := L_Gate_Open;
GVL_COMMAND_SHADOW.G_Wicket_Open := L_Wicket_Open;

// >>> BULK_SYNC_ANCHOR: PRG_Command_Arbitration <<<
          
END_PROGRAM

PROGRAM PRG_PLC_B

            // Вызов основной программы
PRG_System();
// >>> BULK_SYNC_ANCHOR: PRG_PLC_B <<<
          
END_PROGRAM

PROGRAM PRG_Observability_Governor
  VAR
    L_Now_MS : UDINT;
    L_Runtime_Authority_Valid : BOOL;
    L_Publication_Authority_Valid : BOOL;
    L_Recovery_Authority_Valid : BOOL;
    L_Distributed_Authority_Valid : BOOL;
    L_Final_Projection_Barrier_Valid : BOOL;
  END_VAR

            L_Now_MS := GVL_STATUS.G_System_Time_MS;

GVL_OBSERVABILITY_AUTHORITY.Runtime_Failure_Visible := FALSE;
GVL_OBSERVABILITY_AUTHORITY.Output_Decay_Visible := FALSE;
GVL_OBSERVABILITY_AUTHORITY.Transport_Failure_Visible := FALSE;
GVL_OBSERVABILITY_AUTHORITY.Recovery_Failure_Visible := FALSE;
GVL_OBSERVABILITY_AUTHORITY.Fencing_Failure_Visible := FALSE;
GVL_OBSERVABILITY_AUTHORITY.Monotonic_Failure_Visible := FALSE;

GVL_OBSERVABILITY_AUTHORITY.Distributed_Failure_Visible := FALSE;
GVL_OBSERVABILITY_AUTHORITY.Distributed_Quarantine_Visible := FALSE;
GVL_OBSERVABILITY_AUTHORITY.Peer_Runtime_Stale_Visible := FALSE;
GVL_OBSERVABILITY_AUTHORITY.Peer_Snapshot_Stale_Visible := FALSE;
GVL_OBSERVABILITY_AUTHORITY.Peer_Boot_Mismatch_Visible := FALSE;
GVL_OBSERVABILITY_AUTHORITY.Peer_Fencing_Conflict_Visible := FALSE;
GVL_OBSERVABILITY_AUTHORITY.Peer_Semantic_Continuity_Lost_Visible := FALSE;

GVL_OBSERVABILITY_AUTHORITY.Distributed_Publication_Reconciliation_Visible := FALSE;
GVL_OBSERVABILITY_AUTHORITY.Distributed_Publication_Freeze_Visible := FALSE;
GVL_OBSERVABILITY_AUTHORITY.Distributed_Snapshot_Consistency_Visible := FALSE;
GVL_OBSERVABILITY_AUTHORITY.Peer_Publication_Stale_Visible := FALSE;
GVL_OBSERVABILITY_AUTHORITY.Peer_Publication_Divergence_Visible := FALSE;
GVL_OBSERVABILITY_AUTHORITY.Peer_Publication_Reconciliation_Lost_Visible := FALSE;
GVL_OBSERVABILITY_AUTHORITY.Peer_Snapshot_Not_Immutable_Visible := FALSE;
GVL_OBSERVABILITY_AUTHORITY.Distributed_Immutable_Snapshot_Quarantine_Visible := FALSE;

GVL_OBSERVABILITY_AUTHORITY.Distributed_Commit_Visible := FALSE;
GVL_OBSERVABILITY_AUTHORITY.Distributed_Commit_Quarantine_Visible := FALSE;
GVL_OBSERVABILITY_AUTHORITY.Publication_Prepare_Visible := FALSE;
GVL_OBSERVABILITY_AUTHORITY.Publication_Commit_Visible := FALSE;
GVL_OBSERVABILITY_AUTHORITY.Peer_Commit_Ack_Visible := FALSE;
GVL_OBSERVABILITY_AUTHORITY.Peer_Commit_Mismatch_Visible := FALSE;
GVL_OBSERVABILITY_AUTHORITY.Peer_Commit_Replay_Visible := FALSE;
GVL_OBSERVABILITY_AUTHORITY.Peer_Commit_Missing_Visible := FALSE;
GVL_OBSERVABILITY_AUTHORITY.Commit_Lease_Expired_Visible := FALSE;

GVL_OBSERVABILITY_AUTHORITY.Unsafe_State_Published := FALSE;
GVL_OBSERVABILITY_AUTHORITY.Emergency_Visibility_Required := FALSE;

L_Runtime_Authority_Valid :=
    GVL_RUNTIME_EPOCH.Runtime_Runtime_Barrier_OK
    AND GVL_RUNTIME_SNAPSHOT.Snapshot_Publication_Allowed
    AND GVL_RUNTIME_SNAPSHOT.Snapshot_Copy_Valid
    AND GVL_RUNTIME_SNAPSHOT.Snapshot_Isolation_Valid
    AND NOT GVL_RUNTIME_SNAPSHOT.Snapshot_Mutation_Detected;

L_Publication_Authority_Valid :=
    GVL_OUTPUT_EPOCH.Output_Publication_Allowed
    AND GVL_OUTPUT_EPOCH.Output_Publication_Valid
    AND GVL_OUTPUT_EPOCH.Output_Runtime_Epoch_Valid
    AND NOT GVL_OUTPUT_EPOCH.Output_Lease_Expired
    AND NOT GVL_OUTPUT_EPOCH.Output_Forced_Safe_Decay
    AND GVL_TRANSPORT_FRESHNESS.Transport_Freshness_Valid;

L_Recovery_Authority_Valid :=
    GVL_RECOVERY_GOVERNANCE.Recovery_Governance_Valid
    AND NOT GVL_RECOVERY_GOVERNANCE.Recovery_Quarantine_Active
    AND GVL_CONVERGENCE.Convergence_Release_Allowed;

L_Distributed_Authority_Valid :=
    GVL_DISTRIBUTED_EPOCH.Distributed_Reconciliation_Valid
    AND NOT GVL_DISTRIBUTED_EPOCH.Distributed_Quarantine_Active
    AND GVL_DISTRIBUTED_SNAPSHOT.Distributed_Snapshot_Consistent
    AND GVL_DISTRIBUTED_COMMIT.Distributed_Commit_Valid
    AND GVL_Distributed_Execution_Gates.G_Runtime_Valid;

// Final projection proof barrier.
L_Final_Projection_Barrier_Valid :=
    GVL_COMMAND_VERIFY.PreOutput_Barrier_OK
    AND NOT GVL_COMMAND_VERIFY.PreOutput_Block_IO;

GVL_OBSERVABILITY_AUTHORITY.Publication_Runtime_Valid :=
    L_Runtime_Authority_Valid
    AND L_Publication_Authority_Valid
    AND L_Recovery_Authority_Valid
    AND L_Distributed_Authority_Valid
    AND L_Final_Projection_Barrier_Valid;

IF NOT L_Final_Projection_Barrier_Valid THEN
    GVL_OBSERVABILITY_AUTHORITY.Unsafe_State_Published := TRUE;
    GVL_OBSERVABILITY_AUTHORITY.Emergency_Visibility_Required := TRUE;
END_IF;

IF NOT L_Publication_Authority_Valid THEN
    GVL_OBSERVABILITY_AUTHORITY.Output_Decay_Visible := TRUE;
    GVL_OBSERVABILITY_AUTHORITY.Emergency_Visibility_Required := TRUE;
END_IF;

GVL_OBSERVABILITY_AUTHORITY.Observability_Epoch := GVL_OBSERVABILITY_AUTHORITY.Observability_Epoch + 1;
GVL_OBSERVABILITY_AUTHORITY.Observability_Snapshot_Epoch := GVL_OBSERVABILITY_AUTHORITY.Observability_Snapshot_Epoch + 1;

GVL_OBSERVABILITY_AUTHORITY.Observability_Last_Publication_MS := L_Now_MS;

GVL_OBSERVABILITY_AUTHORITY.Observability_Last_Error_Code := 0;
GVL_OBSERVABILITY_AUTHORITY.Observability_Last_Error_Text := '';
          
END_PROGRAM

PROGRAM PLC_PRG
  VAR
    fbSystemRedundancyOrchestrator : FB_System_Redundancy_Orchestrator;
    fbSystemDiagnostics : FB_System_Diagnostics;
    fbStateReplication : FB_State_Replication;
    fbRedundancyManager : FB_Redundancy_Manager;
    fbPLCHeartbeat : FB_PLC_Heartbeat;
    L_Main_Local_State : ST_System_State_Snapshot;
    L_Main_Remote_State : ST_System_State_Snapshot;
    L_Main_Synced_State : ST_System_State_Snapshot;
    L_Main_State_Updated : BOOL;
    L_Main_PLC_Active : BOOL;
    L_Main_RTT_MS : UDINT;
    L_Main_Loss_Count : UDINT;
    L_Main_Max_RTT : UDINT;
  END_VAR

            PRG_Time_Service();
PRG_Time_Monotonic_Governor();
PRG_System_Init();
PRG_Config_Manager();
PRG_Config_Validation();
PRG_Config_Versioning();
PRG_System_Runtime_Base();

PRG_Temporal_Domain();
PRG_Runtime_Core_Domain();
PRG_Safety_Domain();
PRG_Recovery_Domain();
PRG_Distributed_Domain();
PRG_Verification_Domain();
PRG_Semantic_Commit_Governor();

fbPLCHeartbeat(
    VI_Local_ID := GVL_STATUS.G_PLC_ID,
    VI_System_Time := GVL_STATUS.G_System_Time_MS,
    VI_Remote_Pulse := GVL_IO.DI_Partner_Pulse,
    VI_Remote_Is_Active := GVL_IO.DI_Partner_Active,
    VI_Gateway_Ping_OK := GVL_GATEWAY.G_Gateway_Ping_OK,
    VO_Is_Active => L_Main_PLC_Active,
    VO_RTT_MS => L_Main_RTT_MS,
    VO_Loss_Count => L_Main_Loss_Count,
    VO_Max_RTT => L_Main_Max_RTT
);

fbStateReplication(
    VI_Local_Role := SEL(GVL_STATUS.G_Is_Active_PLC, E_PLC_ROLE.ROLE_STANDBY, E_PLC_ROLE.ROLE_ACTIVE),
    VI_Sync_Req := FALSE,
    VI_Local_State := L_Main_Local_State,
    VI_Remote_State := L_Main_Remote_State,
    VI_System_Time_MS := GVL_STATUS.G_System_Time_MS,
    VO_State_Updated => L_Main_State_Updated,
    VO_Synced_State => L_Main_Synced_State
);

fbRedundancyManager(
    VI_System_Time_MS := GVL_STATUS.G_System_Time_MS,
    VI_Local_PLC_ID := GVL_STATUS.G_PLC_ID,
    VI_Remote_Pulse := GVL_IO.DI_Partner_Pulse,
    VI_Remote_Is_Active := GVL_IO.DI_Partner_Active,
    VI_Gateway_Ping_OK := GVL_GATEWAY.G_Gateway_Ping_OK,
    VI_Local_State := L_Main_Local_State,
    VI_Remote_State := L_Main_Remote_State
);

fbSystemDiagnostics();

fbSystemRedundancyOrchestrator(
    VIO_Local_State := L_Main_Local_State,
    VIO_Remote_State := L_Main_Remote_State
);

PRG_Peer_Heartbeat_Ingestion();
PRG_PLC_Arbitration();
PRG_PLC_Fencing_Governor();
PRG_IO_Read();
PRG_Input_Quality_Read();
PRG_Input_Processing();
PRG_Mode_Manager();
PRG_Presence_Manager();
PRG_Safety();
PRG_Safety_Operator();
PRG_Safety_Shutdown();
PRG_Safety_Recovery();
PRG_System_Intent();
PRG_Security();
PRG_System_Access_Maintenance();
PRG_User_Adapt_Control();
PRG_Behavior_Adapt_Profile();
PRG_Scenario_Engine();
PRG_System_Scenario_Rules();
PRG_System_Evacuation();
PRG_Policy();
PRG_Heating_Policy_Manager();
PRG_Heating_Policy_Observer();
PRG_System_Coordinator();
PRG_Command_Arbitration();
PRG_Modbus_Master();
PRG_Modbus_RTU_Bridge();
PRG_Modbus_RTU_Driver();
PRG_Modbus_RTU_SysCom_Backend();
PRG_Modbus_RTU_SysCom_Transport();
PRG_Modbus_Register_Scan();
PRG_OpenTherm_Transport();
PRG_OpenTherm_Adapter_Status();
PRG_Transport_Freshness_Governor();
PRG_Runtime_Barrier();
PRG_Runtime_Snapshot_Governor();
PRG_Peer_Session_Publication();
PRG_HA_Session_Replication();
PRG_Distributed_Peer_Ingestion();
PRG_Distributed_Epoch_Governor();
PRG_Distributed_Snapshot_Publication();
PRG_Distributed_Snapshot_Ingestion();
PRG_Distributed_Snapshot_Governor();
PRG_Distributed_Runtime_Supervisor();
PRG_Distributed_Commit_Publication();
PRG_Distributed_Commit_Ingestion();
PRG_Distributed_Commit_Governor();
PRG_Distributed_Commit_Observability();
PRG_Semantic_Progress_Governor();
PRG_Convergence_Governor();
PRG_Recovery_Cleanup_Governor();
PRG_Observability_Governor();
PRG_Heating();
PRG_Heating_Supervisory_Publication();
PRG_Ventilation();
PRG_Water_Supervisory_Publication();
PRG_Water_Output_Projection();
PRG_Water();
PRG_Access();
PRG_Lighting();
PRG_Output_Freshness_Governor();
PRG_Physical_Snapshot_Governor();
PRG_Sensor_Consensus_Governor();
PRG_Telemetry_Causality_Governor();
PRG_Physical_Authority_Epoch_Governor();
PRG_Authority_Lineage_Governor();
PRG_Authority_Revocation_Governor();
PRG_Authority_Restoration_Governor();
PRG_PreOutput_Safety_Barrier();
PRG_IO_Write();
PRG_Actuation_Authority_Governor();
PRG_Physical_Transaction_Governor();
PRG_Temporal_Stability_Governor();
PRG_Environmental_Authority_Governor();
PRG_Runtime_Resource_Authority_Governor();
PRG_Semantic_Continuity_Authority_Governor();
PRG_Observability_Truth_Governor();
PRG_Historical_Truth_Governor();
PRG_Global_Authority_Sync_Governor();
PRG_Control_Temporal_Coherence_Governor();
PRG_Actuator_Semantic_Verification_Governor();
PRG_Energy_Causality_Governor();
PRG_Runtime_Sustainability_Governor();
PRG_Semantic_Preservation_Governor();
PRG_Operator_Semantic_Alignment_Governor();
PRG_Semantic_Federation_Governor();
PRG_Compliance_Federation_Governor();
PRG_Forensic_Evidence_Governor();
PRG_Epistemic_Integrity_Governor();
PRG_Meta_Governance_Governor();
PRG_Authority_Provenance_Governor();
PRG_Provenance_Continuity_Governor();
PRG_Trust_Epoch_Monotonicity_Governor();
PRG_Semantic_Epoch_Invariance_Governor();
PRG_Governance_Observer_Consensus_Governor();
PRG_Execution_Projection_Integrity_Governor();
PRG_Governance_Feedback_Integrity_Governor();
PRG_Governance_Validator_Integrity_Governor();
PRG_Governance_Liveness_Integrity_Governor();
PRG_Governance_Publication_Binding_Governor();
PRG_Physical_SafeState_Lattice_Governor();
PRG_CrossDomain_FailSafe_Closure_Governor();
PRG_Deterministic_Recovery_Path_Governor();
PRG_Recovery_Ordering_Integrity_Governor();
PRG_Recovery_Reactivation_Control_Governor();
PRG_Authority_Resurrection_Boundary_Governor();
PRG_Energy_Isolation_Causality_Governor();
PRG_Residual_Energy_State_Governor();
PRG_Power_Domain_Segmentation_Governor();
PRG_Energy_Resurrection_Boundary_Governor();
PRG_Physical_Deadlock_Resolution_Governor();
PRG_Execution_Progress_Causality_Governor();
PRG_Resource_Starvation_Boundary_Governor();
PRG_Distributed_Forward_Progress_Governor();
PRG_Safety_Observability_Truth_Governor();
PRG_Physical_Safety_Projection_Governor();
PRG_Unsafe_Transition_Forensics_Governor();
PRG_Distributed_Safety_Reality_Consensus_Governor();
PRG_Temporal_Causality_Closure_Governor();
PRG_Distributed_Epoch_Linearity_Governor();
PRG_Historical_Ordering_Integrity_Governor();
PRG_Causality_Reversal_Prevention_Governor();
PRG_Passive_Runtime_Verification_Governor();
PRG_Semantic_Drift_Observability_Governor();
PRG_Proof_Continuity_Audit_Governor();
PRG_Runtime_Assumption_Integrity_Governor();
PRG_Runtime_Transition_Validator();
PRG_Operational_Intelligence_Governor();
PRG_Causal_Narrative_Engine();
PRG_Physical_Reality_Validation_Governor();
PRG_Survivability_Intelligence_Governor();
PRG_Runtime_Compression_Governor();
PRG_Runtime_Budget_Governor();
PRG_Controlled_Capability_Shedding_Governor();
PRG_Semantic_Execution_Control_Governor();
PRG_Industrial_Maintainability_Governor();
PRG_Observability_Authority_Governor();
PRG_Command_Verifier();
PRG_Explainability();
PRG_System_Health();
PRG_System_Alarm_Gateway();
PRG_System_Diagnostics();
PRG_System_Diagnostics_Ext();
PRG_System_History();
PRG_System_BlackBox();
PRG_System_Trend();
PRG_System_Simulation();
PRG_HMI_Dashboard();
PRG_Debug_View();

// >>> BULK_SYNC_ANCHOR: MAIN <<<
          
END_PROGRAM
